LIN {X 0,Y 539.33,Z 456.687,A -85,B 0,C 180,E1 -4153.302,E2 -4153.302} C_VEL
LIN {X 0,Y 539.491,Z 386.193,A -85,B 0,C 180,E1 -4154.273,E2 -4154.273} C_VEL
LIN {X 0,Y 538.254,Z 382.203,A -85,B 0,C 180,E1 -4154.395,E2 -4154.395} C_VEL
LIN {X 0,Y 538.117,Z 381.5,A -85,B 0,C 180,E1 -4154.551,E2 -4154.551} C_VEL
LIN {X 0,Y 538.039,Z 381.463,A -85,B 0,C 180,E1 -4157.532,E2 -4157.532} C_VEL
LIN {X 0,Y 538.041,Z 381.467,A -85,B 0,C 180,E1 -4160.651,E2 -4160.651} C_VEL
LIN {X 0,Y 538.006,Z 381.464,A -85,B 0,C 180,E1 -4163.888,E2 -4163.888} C_VEL
LIN {X 0,Y 538.039,Z 381.463,A -85,B 0,C 180,E1 -4166.367,E2 -4166.367} C_VEL
LIN {X 0,Y 538.01,Z 381.462,A -85,B 0,C 180,E1 -4169.392,E2 -4169.392} C_VEL
LIN {X 0,Y 537.341,Z 381.546,A -85,B 0,C 180,E1 -4170.017,E2 -4170.017} C_VEL
LIN {X 0,Y 534.471,Z 381.909,A -85,B 0,C 180,E1 -4171.03,E2 -4171.03} C_VEL
LIN {X 0,Y 532.057,Z 382.207,A -85,B 0,C 180,E1 -4171.846,E2 -4171.846} C_VEL
LIN {X 0,Y 531.035,Z 382.338,A -85,B 0,C 180,E1 -4172.476,E2 -4172.476} C_VEL
LIN {X 0,Y 530.96,Z 382.343,A -85,B 0,C 180,E1 -4172.689,E2 -4172.689} C_VEL
LIN {X 0,Y 530.953,Z 382.342,A -85,B 0,C 180,E1 -4175.62,E2 -4175.62} C_VEL
LIN {X 0,Y 530.967,Z 382.346,A -85,B 0,C 180,E1 -4178.653,E2 -4178.653} C_VEL
LIN {X 0,Y 530.992,Z 382.337,A -85,B 0,C 180,E1 -4181.436,E2 -4181.436} C_VEL
LIN {X 0,Y 530.97,Z 382.348,A -85,B 0,C 180,E1 -4184.549,E2 -4184.549} C_VEL
LIN {X 0,Y 530.975,Z 382.34,A -85,B 0,C 180,E1 -4187.836,E2 -4187.836} C_VEL
LIN {X 0,Y 530.974,Z 382.343,A -85,B 0,C 180,E1 -4190.555,E2 -4190.555} C_VEL
LIN {X 0,Y 530.953,Z 382.344,A -85,B 0,C 180,E1 -4193.441,E2 -4193.441} C_VEL
LIN {X 0,Y 531.002,Z 382.345,A -85,B 0,C 180,E1 -4196.494,E2 -4196.494} C_VEL
LIN {X 0,Y 530.969,Z 382.342,A -85,B 0,C 180,E1 -4199.357,E2 -4199.357} C_VEL
LIN {X 0,Y 531.024,Z 382.51,A -85,B 0,C 180,E1 -4202.212,E2 -4202.212} C_VEL
LIN {X 0,Y 533.353,Z 393.17,A -85,B 0,C 180,E1 -4203.642,E2 -4203.642} C_VEL
LIN {X 0,Y 533.057,Z 413.258,A -85,B 0,C 180,E1 -4206.083,E2 -4206.083} C_VEL
LIN {X 0,Y 532.641,Z 436.75,A -85,B 0,C 180,E1 -4208.927,E2 -4208.927} C_VEL
LIN {X 0,Y 532.055,Z 463.536,A -85,B 0,C 180,E1 -4212.135,E2 -4212.135} C_VEL
LIN {X 0,Y 531.666,Z 488.086,A -85,B 0,C 180,E1 -4215.055,E2 -4215.055} C_VEL
LIN {X 0,Y 532.804,Z 497.302,A -85,B 0,C 180,E1 -4215.24,E2 -4215.24} C_VEL
LIN {X 0,Y 532.44,Z 598.014,A -85,B 0,C 180,E1 -4216.62,E2 -4216.62} C_VEL
LIN {X 0,Y 532.274,Z 610.527,A -85,B 0,C 180,E1 -4216.932,E2 -4216.932} C_VEL
LIN {X 0,Y 532.051,Z 622.317,A -85,B 0,C 180,E1 -4217.363,E2 -4217.363} C_VEL
LIN {X 0,Y 531.805,Z 635.2,A -85,B 0,C 180,E1 -4218.006,E2 -4218.006} C_VEL
LIN {X 0,Y 531.57,Z 646.587,A -85,B 0,C 180,E1 -4218.755,E2 -4218.755} C_VEL
LIN {X 0,Y 531.283,Z 655.996,A -85,B 0,C 180,E1 -4219.52,E2 -4219.52} C_VEL
LIN {X 0,Y 531.121,Z 663.859,A -85,B 0,C 180,E1 -4220.287,E2 -4220.287} C_VEL
LIN {X 0,Y 530.936,Z 670.557,A -85,B 0,C 180,E1 -4221.052,E2 -4221.052} C_VEL
LIN {X 0,Y 530.785,Z 677.606,A -85,B 0,C 180,E1 -4222.008,E2 -4222.008} C_VEL
LIN {X 0,Y 530.671,Z 683.5,A -85,B 0,C 180,E1 -4222.963,E2 -4222.963} C_VEL
LIN {X 0,Y 530.607,Z 688.403,A -85,B 0,C 180,E1 -4223.917,E2 -4223.917} C_VEL
LIN {X 0,Y 530.459,Z 693.137,A -85,B 0,C 180,E1 -4225.06,E2 -4225.06} C_VEL
LIN {X 0,Y 530.516,Z 696.771,A -85,B 0,C 180,E1 -4226.202,E2 -4226.202} C_VEL
LIN {X 0,Y 530.411,Z 700.139,A -85,B 0,C 180,E1 -4227.722,E2 -4227.722} C_VEL
LIN {X 0,Y 530.344,Z 701.716,A -85,B 0,C 180,E1 -4229.241,E2 -4229.241} C_VEL
LIN {X 0,Y 530.343,Z 701.997,A -85,B 0,C 180,E1 -4230,E2 -4230} C_VEL
LIN {X 0,Y 530.361,Z 701.19,A -85,B 0,C 180,E1 -4231.519,E2 -4231.519} C_VEL
LIN {X 0,Y 530.411,Z 700.285,A -85,B 0,C 180,E1 -4232.278,E2 -4232.278} C_VEL
LIN {X 0,Y 530.516,Z 697.021,A -85,B 0,C 180,E1 -4233.798,E2 -4233.798} C_VEL
LIN {X 0,Y 530.458,Z 693.464,A -85,B 0,C 180,E1 -4234.94,E2 -4234.94} C_VEL
LIN {X 0,Y 530.582,Z 688.812,A -85,B 0,C 180,E1 -4236.083,E2 -4236.083} C_VEL
LIN {X 0,Y 530.628,Z 683.999,A -85,B 0,C 180,E1 -4237.037,E2 -4237.037} C_VEL
LIN {X 0,Y 530.772,Z 678.202,A -85,B 0,C 180,E1 -4237.992,E2 -4237.992} C_VEL
LIN {X 0,Y 530.9,Z 671.262,A -85,B 0,C 180,E1 -4238.949,E2 -4238.949} C_VEL
LIN {X 0,Y 531.09,Z 664.693,A -85,B 0,C 180,E1 -4239.714,E2 -4239.714} C_VEL
LIN {X 0,Y 531.31,Z 655.926,A -85,B 0,C 180,E1 -4240.576,E2 -4240.576} C_VEL
LIN {X 0,Y 531.599,Z 645.228,A -85,B 0,C 180,E1 -4241.438,E2 -4241.438} C_VEL
LIN {X 0,Y 531.847,Z 633.026,A -85,B 0,C 180,E1 -4242.206,E2 -4242.206} C_VEL
LIN {X 0,Y 532.074,Z 620.98,A -85,B 0,C 180,E1 -4242.782,E2 -4242.782} C_VEL
LIN {X 0,Y 532.26,Z 608.699,A -85,B 0,C 180,E1 -4243.215,E2 -4243.215} C_VEL
LIN {X 0,Y 532.463,Z 596.37,A -85,B 0,C 180,E1 -4243.501,E2 -4243.501} C_VEL
LIN {X 0,Y 532.768,Z 496.104,A -85,B 0,C 180,E1 -4244.868,E2 -4244.868} C_VEL
LIN {X 0,Y 531.685,Z 488.274,A -85,B 0,C 180,E1 -4245.02,E2 -4245.02} C_VEL
LIN {X 0,Y 532.074,Z 463.132,A -85,B 0,C 180,E1 -4248.005,E2 -4248.005} C_VEL
LIN {X 0,Y 532.617,Z 437.549,A -85,B 0,C 180,E1 -4251.074,E2 -4251.074} C_VEL
LIN {X 0,Y 533.063,Z 414.001,A -85,B 0,C 180,E1 -4253.917,E2 -4253.917} C_VEL
LIN {X 0,Y 533.411,Z 393.872,A -85,B 0,C 180,E1 -4256.37,E2 -4256.37} C_VEL
LIN {X 0,Y 531.004,Z 382.431,A -85,B 0,C 180,E1 -4257.907,E2 -4257.907} C_VEL
LIN {X 0,Y 530.955,Z 382.348,A -85,B 0,C 180,E1 -4261.08,E2 -4261.08} C_VEL
LIN {X 0,Y 530.967,Z 382.346,A -85,B 0,C 180,E1 -4263.775,E2 -4263.775} C_VEL
LIN {X 0,Y 530.919,Z 382.344,A -85,B 0,C 180,E1 -4266.562,E2 -4266.562} C_VEL
LIN {X 0,Y 530.985,Z 382.345,A -85,B 0,C 180,E1 -4269.444,E2 -4269.444} C_VEL
LIN {X 0,Y 530.917,Z 382.348,A -85,B 0,C 180,E1 -4272.463,E2 -4272.463} C_VEL
LIN {X 0,Y 530.969,Z 382.339,A -85,B 0,C 180,E1 -4275.451,E2 -4275.451} C_VEL
LIN {X 0,Y 530.963,Z 382.341,A -85,B 0,C 180,E1 -4278.561,E2 -4278.561} C_VEL
LIN {X 0,Y 530.954,Z 382.35,A -85,B 0,C 180,E1 -4281.529,E2 -4281.529} C_VEL
LIN {X 0,Y 530.938,Z 382.345,A -85,B 0,C 180,E1 -4284.378,E2 -4284.378} C_VEL
LIN {X 0,Y 530.97,Z 382.338,A -85,B 0,C 180,E1 -4287.133,E2 -4287.133} C_VEL
LIN {X 0,Y 530.952,Z 382.348,A -85,B 0,C 180,E1 -4289.802,E2 -4289.802} C_VEL
LIN {X 0,Y 530.959,Z 382.342,A -85,B 0,C 180,E1 -4292.48,E2 -4292.48} C_VEL
LIN {X 0,Y 530.953,Z 382.342,A -85,B 0,C 180,E1 -4294.94,E2 -4294.94} C_VEL
LIN {X 0,Y 530.981,Z 382.345,A -85,B 0,C 180,E1 -4297.898,E2 -4297.898} C_VEL
LIN {X 0,Y 530.973,Z 382.338,A -85,B 0,C 180,E1 -4300.676,E2 -4300.676} C_VEL
LIN {X 0,Y 530.942,Z 382.34,A -85,B 0,C 180,E1 -4303.069,E2 -4303.069} C_VEL
LIN {X 0,Y 531.012,Z 382.34,A -85,B 0,C 180,E1 -4305.436,E2 -4305.436} C_VEL
LIN {X 0,Y 530.99,Z 382.331,A -85,B 0,C 180,E1 -4308.549,E2 -4308.549} C_VEL
LIN {X 0,Y 530.993,Z 382.344,A -85,B 0,C 180,E1 -4311.628,E2 -4311.628} C_VEL
LIN {X 0,Y 531.088,Z 382.32,A -85,B 0,C 180,E1 -4314.685,E2 -4314.685} C_VEL
LIN {X 0,Y 531.136,Z 382.325,A -85,B 0,C 180,E1 -4317.725,E2 -4317.725} C_VEL
LIN {X 0,Y 531.131,Z 382.324,A -85,B 0,C 180,E1 -4320,E2 -4320} C_VEL
LIN {X 0,Y 531.136,Z 382.315,A -85,B 0,C 180,E1 -4322.275,E2 -4322.275} C_VEL
LIN {X 0,Y 531.085,Z 382.327,A -85,B 0,C 180,E1 -4325.315,E2 -4325.315} C_VEL
LIN {X 0,Y 530.986,Z 382.335,A -85,B 0,C 180,E1 -4328.372,E2 -4328.372} C_VEL
LIN {X 0,Y 531.015,Z 382.338,A -85,B 0,C 180,E1 -4331.65,E2 -4331.65} C_VEL
LIN {X 0,Y 530.967,Z 382.339,A -85,B 0,C 180,E1 -4334.928,E2 -4334.928} C_VEL
LIN {X 0,Y 530.973,Z 382.342,A -85,B 0,C 180,E1 -4337.724,E2 -4337.724} C_VEL
LIN {X 0,Y 530.939,Z 382.343,A -85,B 0,C 180,E1 -4340.94,E2 -4340.94} C_VEL
LIN {X 0,Y 530.952,Z 382.34,A -85,B 0,C 180,E1 -4343.397,E2 -4343.397} C_VEL
LIN {X 0,Y 530.93,Z 382.353,A -85,B 0,C 180,E1 -4345.902,E2 -4345.902} C_VEL
LIN {X 0,Y 530.932,Z 382.341,A -85,B 0,C 180,E1 -4348.459,E2 -4348.459} C_VEL
LIN {X 0,Y 530.946,Z 382.343,A -85,B 0,C 180,E1 -4351.08,E2 -4351.08} C_VEL
LIN {X 0,Y 530.952,Z 382.348,A -85,B 0,C 180,E1 -4353.775,E2 -4353.775} C_VEL
LIN {X 0,Y 530.908,Z 382.349,A -85,B 0,C 180,E1 -4356.562,E2 -4356.562} C_VEL
LIN {X 0,Y 530.94,Z 382.344,A -85,B 0,C 180,E1 -4359.448,E2 -4359.448} C_VEL
LIN {X 0,Y 530.906,Z 382.344,A -85,B 0,C 180,E1 -4362.464,E2 -4362.464} C_VEL
LIN {X 0,Y 530.963,Z 382.344,A -85,B 0,C 180,E1 -4365.45,E2 -4365.45} C_VEL
LIN {X 0,Y 530.91,Z 382.337,A -85,B 0,C 180,E1 -4368.556,E2 -4368.556} C_VEL
LIN {X 0,Y 530.932,Z 382.348,A -85,B 0,C 180,E1 -4371.527,E2 -4371.527} C_VEL
LIN {X 0,Y 530.927,Z 382.35,A -85,B 0,C 180,E1 -4374.377,E2 -4374.377} C_VEL
LIN {X 0,Y 530.946,Z 382.345,A -85,B 0,C 180,E1 -4377.132,E2 -4377.132} C_VEL
LIN {X 0,Y 530.934,Z 382.353,A -85,B 0,C 180,E1 -4379.8,E2 -4379.8} C_VEL
LIN {X 0,Y 531.006,Z 382.538,A -85,B 0,C 180,E1 -4381.519,E2 -4381.519} C_VEL
LIN {X 0,Y 533.419,Z 393.223,A -85,B 0,C 180,E1 -4382.964,E2 -4382.964} C_VEL
LIN {X 0,Y 533.514,Z 400.976,A -85,B 0,C 180,E1 -4383.902,E2 -4383.902} C_VEL
LIN {X 0,Y 532.934,Z 426.254,A -85,B 0,C 180,E1 -4386.901,E2 -4386.901} C_VEL
LIN {X 0,Y 532.347,Z 450.23,A -85,B 0,C 180,E1 -4389.714,E2 -4389.714} C_VEL
LIN {X 0,Y 531.914,Z 476.387,A -85,B 0,C 180,E1 -4392.705,E2 -4392.705} C_VEL
LIN {X 0,Y 531.617,Z 496.923,A -85,B 0,C 180,E1 -4395.02,E2 -4395.02} C_VEL
LIN {X 0,Y 532.795,Z 507.185,A -85,B 0,C 180,E1 -4395.211,E2 -4395.211} C_VEL
LIN {X 0,Y 532.377,Z 607.666,A -85,B 0,C 180,E1 -4396.594,E2 -4396.594} C_VEL
LIN {X 0,Y 532.181,Z 620.892,A -85,B 0,C 180,E1 -4396.929,E2 -4396.929} C_VEL
LIN {X 0,Y 531.981,Z 633.67,A -85,B 0,C 180,E1 -4397.409,E2 -4397.409} C_VEL
LIN {X 0,Y 531.756,Z 645.607,A -85,B 0,C 180,E1 -4398.019,E2 -4398.019} C_VEL
LIN {X 0,Y 531.508,Z 656.848,A -85,B 0,C 180,E1 -4398.753,E2 -4398.753} C_VEL
LIN {X 0,Y 531.224,Z 667.468,A -85,B 0,C 180,E1 -4399.615,E2 -4399.615} C_VEL
LIN {X 0,Y 531.062,Z 676.091,A -85,B 0,C 180,E1 -4400.478,E2 -4400.478} C_VEL
LIN {X 0,Y 530.887,Z 683.959,A -85,B 0,C 180,E1 -4401.435,E2 -4401.435} C_VEL
LIN {X 0,Y 530.685,Z 691.62,A -85,B 0,C 180,E1 -4402.581,E2 -4402.581} C_VEL
LIN {X 0,Y 530.604,Z 698.678,A -85,B 0,C 180,E1 -4403.917,E2 -4403.917} C_VEL
LIN {X 0,Y 530.459,Z 703.372,A -85,B 0,C 180,E1 -4405.06,E2 -4405.06} C_VEL
LIN {X 0,Y 530.516,Z 706.957,A -85,B 0,C 180,E1 -4406.202,E2 -4406.202} C_VEL
LIN {X 0,Y 530.457,Z 708.806,A -85,B 0,C 180,E1 -4406.962,E2 -4406.962} C_VEL
LIN {X 0,Y 530.411,Z 710.193,A -85,B 0,C 180,E1 -4407.722,E2 -4407.722} C_VEL
LIN {X 0,Y 530.344,Z 711.785,A -85,B 0,C 180,E1 -4409.241,E2 -4409.241} C_VEL
LIN {X 0,Y 530.342,Z 712,A -85,B 0,C 180,E1 -4410,E2 -4410} C_VEL
LIN {X 0,Y 530.361,Z 711.183,A -85,B 0,C 180,E1 -4411.519,E2 -4411.519} C_VEL
LIN {X 0,Y 530.411,Z 710.196,A -85,B 0,C 180,E1 -4412.278,E2 -4412.278} C_VEL
LIN {X 0,Y 530.457,Z 708.81,A -85,B 0,C 180,E1 -4413.038,E2 -4413.038} C_VEL
LIN {X 0,Y 530.522,Z 705.895,A -85,B 0,C 180,E1 -4414.178,E2 -4414.178} C_VEL
LIN {X 0,Y 530.524,Z 701.948,A -85,B 0,C 180,E1 -4415.321,E2 -4415.321} C_VEL
LIN {X 0,Y 530.599,Z 696.262,A -85,B 0,C 180,E1 -4416.582,E2 -4416.582} C_VEL
LIN {X 0,Y 530.758,Z 689.235,A -85,B 0,C 180,E1 -4417.8,E2 -4417.8} C_VEL
LIN {X 0,Y 530.93,Z 680.992,A -85,B 0,C 180,E1 -4418.948,E2 -4418.948} C_VEL
LIN {X 0,Y 531.139,Z 672.486,A -85,B 0,C 180,E1 -4419.905,E2 -4419.905} C_VEL
LIN {X 0,Y 531.376,Z 661.842,A -85,B 0,C 180,E1 -4420.864,E2 -4420.864} C_VEL
LIN {X 0,Y 531.653,Z 650.613,A -85,B 0,C 180,E1 -4421.672,E2 -4421.672} C_VEL
LIN {X 0,Y 531.885,Z 639.604,A -85,B 0,C 180,E1 -4422.302,E2 -4422.302} C_VEL
LIN {X 0,Y 532.09,Z 627.599,A -85,B 0,C 180,E1 -4422.83,E2 -4422.83} C_VEL
LIN {X 0,Y 532.26,Z 613.764,A -85,B 0,C 180,E1 -4423.263,E2 -4423.263} C_VEL
LIN {X 0,Y 532.443,Z 599.688,A -85,B 0,C 180,E1 -4423.526,E2 -4423.526} C_VEL
LIN {X 0,Y 532.667,Z 505.458,A -85,B 0,C 180,E1 -4424.808,E2 -4424.808} C_VEL
LIN {X 0,Y 531.577,Z 496.346,A -85,B 0,C 180,E1 -4424.981,E2 -4424.981} C_VEL
LIN {X 0,Y 531.934,Z 469.551,A -85,B 0,C 180,E1 -4427.959,E2 -4427.959} C_VEL
LIN {X 0,Y 532.362,Z 443.563,A -85,B 0,C 180,E1 -4430.882,E2 -4430.882} C_VEL
LIN {X 0,Y 532.768,Z 416.948,A -85,B 0,C 180,E1 -4433.931,E2 -4433.931} C_VEL
LIN {X 0,Y 533.15,Z 393.927,A -85,B 0,C 180,E1 -4436.628,E2 -4436.628} C_VEL
LIN {X 0,Y 531.08,Z 383.141,A -85,B 0,C 180,E1 -4438.02,E2 -4438.02} C_VEL
LIN {X 0,Y 530.966,Z 382.478,A -85,B 0,C 180,E1 -4438.134,E2 -4438.134} C_VEL
LIN {X 0,Y 530.936,Z 382.349,A -85,B 0,C 180,E1 -4441.081,E2 -4441.081} C_VEL
LIN {X 0,Y 530.934,Z 382.353,A -85,B 0,C 180,E1 -4443.777,E2 -4443.777} C_VEL
LIN {X 0,Y 530.906,Z 382.351,A -85,B 0,C 180,E1 -4446.563,E2 -4446.563} C_VEL
LIN {X 0,Y 530.94,Z 382.349,A -85,B 0,C 180,E1 -4449.448,E2 -4449.448} C_VEL
LIN {X 0,Y 530.912,Z 382.35,A -85,B 0,C 180,E1 -4452.463,E2 -4452.463} C_VEL
LIN {X 0,Y 530.965,Z 382.347,A -85,B 0,C 180,E1 -4455.451,E2 -4455.451} C_VEL
LIN {X 0,Y 530.957,Z 382.342,A -85,B 0,C 180,E1 -4458.561,E2 -4458.561} C_VEL
LIN {X 0,Y 530.953,Z 382.351,A -85,B 0,C 180,E1 -4461.529,E2 -4461.529} C_VEL
LIN {X 0,Y 530.949,Z 382.345,A -85,B 0,C 180,E1 -4464.379,E2 -4464.379} C_VEL
LIN {X 0,Y 530.969,Z 382.345,A -85,B 0,C 180,E1 -4467.133,E2 -4467.133} C_VEL
LIN {X 0,Y 530.971,Z 382.346,A -85,B 0,C 180,E1 -4469.803,E2 -4469.803} C_VEL
LIN {X 0,Y 530.969,Z 382.341,A -85,B 0,C 180,E1 -4472.477,E2 -4472.477} C_VEL
LIN {X 0,Y 530.981,Z 382.342,A -85,B 0,C 180,E1 -4474.941,E2 -4474.941} C_VEL
LIN {X 0,Y 530.974,Z 382.342,A -85,B 0,C 180,E1 -4478.247,E2 -4478.247} C_VEL
LIN {X 0,Y 530.996,Z 382.341,A -85,B 0,C 180,E1 -4480.677,E2 -4480.677} C_VEL
LIN {X 0,Y 530.978,Z 382.348,A -85,B 0,C 180,E1 -4483.071,E2 -4483.071} C_VEL
LIN {X 0,Y 531.093,Z 382.456,A -85,B 0,C 180,E1 -4485.405,E2 -4485.405} C_VEL
LIN {X 0,Y 531.258,Z 383.232,A -85,B 0,C 180,E1 -4485.528,E2 -4485.528} C_VEL
LIN {X 0,Y 532.723,Z 388.293,A -85,B 0,C 180,E1 -4485.664,E2 -4485.664} C_VEL
LIN {X 0,Y 532.338,Z 463.302,A -85,B 0,C 180,E1 -4486.739,E2 -4486.739} C_VEL
LIN {X 0,Y 532.281,Z 476.373,A -85,B 0,C 180,E1 -4487.077,E2 -4487.077} C_VEL
LIN {X 0,Y 532.153,Z 488.956,A -85,B 0,C 180,E1 -4487.559,E2 -4487.559} C_VEL
LIN {X 0,Y 531.944,Z 500.739,A -85,B 0,C 180,E1 -4488.173,E2 -4488.173} C_VEL
LIN {X 0,Y 531.755,Z 512.234,A -85,B 0,C 180,E1 -4488.951,E2 -4488.951} C_VEL
LIN {X 0,Y 531.533,Z 522.416,A -85,B 0,C 180,E1 -4489.814,E2 -4489.814} C_VEL
LIN {X 0,Y 531.339,Z 530.703,A -85,B 0,C 180,E1 -4490.675,E2 -4490.675} C_VEL
LIN {X 0,Y 531.143,Z 539.63,A -85,B 0,C 180,E1 -4491.822,E2 -4491.822} C_VEL
LIN {X 0,Y 531.01,Z 545.698,A -85,B 0,C 180,E1 -4492.777,E2 -4492.777} C_VEL
LIN {X 0,Y 530.92,Z 551.605,A -85,B 0,C 180,E1 -4493.921,E2 -4493.921} C_VEL
LIN {X 0,Y 530.758,Z 556.277,A -85,B 0,C 180,E1 -4495.062,E2 -4495.062} C_VEL
LIN {X 0,Y 530.707,Z 559.862,A -85,B 0,C 180,E1 -4496.203,E2 -4496.203} C_VEL
LIN {X 0,Y 530.688,Z 561.676,A -85,B 0,C 180,E1 -4496.963,E2 -4496.963} C_VEL
LIN {X 0,Y 530.612,Z 563.086,A -85,B 0,C 180,E1 -4497.723,E2 -4497.723} C_VEL
LIN {X 0,Y 530.593,Z 564.638,A -85,B 0,C 180,E1 -4499.241,E2 -4499.241} C_VEL
LIN {X 0,Y 530.583,Z 564.855,A -85,B 0,C 180,E1 -4500,E2 -4500} C_VEL
LIN {X 0,Y 530.575,Z 564.046,A -85,B 0,C 180,E1 -4501.518,E2 -4501.518} C_VEL
LIN {X 0,Y 530.607,Z 563.084,A -85,B 0,C 180,E1 -4502.277,E2 -4502.277} C_VEL
LIN {X 0,Y 530.643,Z 561.706,A -85,B 0,C 180,E1 -4503.037,E2 -4503.037} C_VEL
LIN {X 0,Y 530.709,Z 557.643,A -85,B 0,C 180,E1 -4504.557,E2 -4504.557} C_VEL
LIN {X 0,Y 530.811,Z 553.379,A -85,B 0,C 180,E1 -4505.699,E2 -4505.699} C_VEL
LIN {X 0,Y 530.884,Z 547.935,A -85,B 0,C 180,E1 -4506.843,E2 -4506.843} C_VEL
LIN {X 0,Y 531.03,Z 541.097,A -85,B 0,C 180,E1 -4507.988,E2 -4507.988} C_VEL
LIN {X 0,Y 531.24,Z 534.11,A -85,B 0,C 180,E1 -4508.943,E2 -4508.943} C_VEL
LIN {X 0,Y 531.382,Z 525.669,A -85,B 0,C 180,E1 -4509.901,E2 -4509.901} C_VEL
LIN {X 0,Y 531.633,Z 515.231,A -85,B 0,C 180,E1 -4510.858,E2 -4510.858} C_VEL
LIN {X 0,Y 531.924,Z 503.763,A -85,B 0,C 180,E1 -4511.695,E2 -4511.695} C_VEL
LIN {X 0,Y 532.036,Z 493.307,A -85,B 0,C 180,E1 -4512.299,E2 -4512.299} C_VEL
LIN {X 0,Y 532.194,Z 481.358,A -85,B 0,C 180,E1 -4512.828,E2 -4512.828} C_VEL
LIN {X 0,Y 532.31,Z 468.412,A -85,B 0,C 180,E1 -4513.238,E2 -4513.238} C_VEL
LIN {X 0,Y 532.418,Z 454.629,A -85,B 0,C 180,E1 -4513.502,E2 -4513.502} C_VEL
LIN {X 0,Y 532.598,Z 387.511,A -85,B 0,C 180,E1 -4514.443,E2 -4514.443} C_VEL
LIN {X 0,Y 531.213,Z 383.1,A -85,B 0,C 180,E1 -4514.575,E2 -4514.575} C_VEL
LIN {X 0,Y 531.049,Z 382.389,A -85,B 0,C 180,E1 -4514.729,E2 -4514.729} C_VEL
LIN {X 0,Y 530.985,Z 382.341,A -85,B 0,C 180,E1 -4517.724,E2 -4517.724} C_VEL
LIN {X 0,Y 531.028,Z 382.336,A -85,B 0,C 180,E1 -4520.127,E2 -4520.127} C_VEL
LIN {X 0,Y 530.949,Z 382.35,A -85,B 0,C 180,E1 -4522.573,E2 -4522.573} C_VEL
LIN {X 0,Y 531.002,Z 382.341,A -85,B 0,C 180,E1 -4525.058,E2 -4525.058} C_VEL
LIN {X 0,Y 530.973,Z 382.338,A -85,B 0,C 180,E1 -4527.598,E2 -4527.598} C_VEL
LIN {X 0,Y 530.972,Z 382.34,A -85,B 0,C 180,E1 -4530.197,E2 -4530.197} C_VEL
LIN {X 0,Y 530.96,Z 382.343,A -85,B 0,C 180,E1 -4532.689,E2 -4532.689} C_VEL
LIN {X 0,Y 530.309,Z 382.426,A -85,B 0,C 180,E1 -4533.322,E2 -4533.322} C_VEL
LIN {X 0,Y 527.435,Z 382.783,A -85,B 0,C 180,E1 -4534.349,E2 -4534.349} C_VEL
LIN {X 0,Y 525.002,Z 383.086,A -85,B 0,C 180,E1 -4535.176,E2 -4535.176} C_VEL
LIN {X 0,Y 523.969,Z 383.213,A -85,B 0,C 180,E1 -4535.816,E2 -4535.816} C_VEL
LIN {X 0,Y 523.893,Z 383.223,A -85,B 0,C 180,E1 -4536.032,E2 -4536.032} C_VEL
LIN {X 0,Y 523.922,Z 383.222,A -85,B 0,C 180,E1 -4539.085,E2 -4539.085} C_VEL
LIN {X 0,Y 523.943,Z 383.216,A -85,B 0,C 180,E1 -4542.12,E2 -4542.12} C_VEL
LIN {X 0,Y 523.943,Z 383.216,A -85,B 0,C 180,E1 -4545.311,E2 -4545.311} C_VEL
LIN {X 0,Y 523.956,Z 383.222,A -85,B 0,C 180,E1 -4548.69,E2 -4548.69} C_VEL
LIN {X 0,Y 523.915,Z 383.215,A -85,B 0,C 180,E1 -4551.898,E2 -4551.898} C_VEL
LIN {X 0,Y 523.925,Z 383.219,A -85,B 0,C 180,E1 -4554.912,E2 -4554.912} C_VEL
LIN {X 0,Y 523.938,Z 383.215,A -85,B 0,C 180,E1 -4557.68,E2 -4557.68} C_VEL
LIN {X 0,Y 523.955,Z 383.223,A -85,B 0,C 180,E1 -4560.677,E2 -4560.677} C_VEL
LIN {X 0,Y 523.987,Z 383.416,A -85,B 0,C 180,E1 -4562.002,E2 -4562.002} C_VEL
LIN {X 0,Y 526.586,Z 395.433,A -85,B 0,C 180,E1 -4563.615,E2 -4563.615} C_VEL
LIN {X 0,Y 526.099,Z 419.563,A -85,B 0,C 180,E1 -4566.583,E2 -4566.583} C_VEL
LIN {X 0,Y 525.542,Z 443.703,A -85,B 0,C 180,E1 -4569.527,E2 -4569.527} C_VEL
LIN {X 0,Y 525.009,Z 468.06,A -85,B 0,C 180,E1 -4572.471,E2 -4572.471} C_VEL
LIN {X 0,Y 524.739,Z 488.377,A -85,B 0,C 180,E1 -4574.873,E2 -4574.873} C_VEL
LIN {X 0,Y 525.966,Z 498.434,A -85,B 0,C 180,E1 -4575.059,E2 -4575.059} C_VEL
LIN {X 0,Y 525.54,Z 597.969,A -85,B 0,C 180,E1 -4576.441,E2 -4576.441} C_VEL
LIN {X 0,Y 525.372,Z 610.614,A -85,B 0,C 180,E1 -4576.757,E2 -4576.757} C_VEL
LIN {X 0,Y 525.091,Z 623.487,A -85,B 0,C 180,E1 -4577.242,E2 -4577.242} C_VEL
LIN {X 0,Y 524.827,Z 636.17,A -85,B 0,C 180,E1 -4577.9,E2 -4577.9} C_VEL
LIN {X 0,Y 524.605,Z 646.702,A -85,B 0,C 180,E1 -4578.603,E2 -4578.603} C_VEL
LIN {X 0,Y 524.274,Z 657.16,A -85,B 0,C 180,E1 -4579.476,E2 -4579.476} C_VEL
LIN {X 0,Y 524.004,Z 667.467,A -85,B 0,C 180,E1 -4580.544,E2 -4580.544} C_VEL
LIN {X 0,Y 523.767,Z 676.422,A -85,B 0,C 180,E1 -4581.706,E2 -4581.706} C_VEL
LIN {X 0,Y 523.61,Z 683.596,A -85,B 0,C 180,E1 -4582.868,E2 -4582.868} C_VEL
LIN {X 0,Y 523.518,Z 688.478,A -85,B 0,C 180,E1 -4583.835,E2 -4583.835} C_VEL
LIN {X 0,Y 523.383,Z 693.192,A -85,B 0,C 180,E1 -4584.993,E2 -4584.993} C_VEL
LIN {X 0,Y 523.443,Z 696.815,A -85,B 0,C 180,E1 -4586.151,E2 -4586.151} C_VEL
LIN {X 0,Y 523.368,Z 698.695,A -85,B 0,C 180,E1 -4586.921,E2 -4586.921} C_VEL
LIN {X 0,Y 523.335,Z 700.161,A -85,B 0,C 180,E1 -4587.691,E2 -4587.691} C_VEL
LIN {X 0,Y 523.25,Z 701.746,A -85,B 0,C 180,E1 -4589.231,E2 -4589.231} C_VEL
LIN {X 0,Y 523.247,Z 702.013,A -85,B 0,C 180,E1 -4590,E2 -4590} C_VEL
LIN {X 0,Y 523.275,Z 701.22,A -85,B 0,C 180,E1 -4591.539,E2 -4591.539} C_VEL
LIN {X 0,Y 523.335,Z 700.298,A -85,B 0,C 180,E1 -4592.309,E2 -4592.309} C_VEL
LIN {X 0,Y 523.444,Z 697.06,A -85,B 0,C 180,E1 -4593.849,E2 -4593.849} C_VEL
LIN {X 0,Y 523.383,Z 693.514,A -85,B 0,C 180,E1 -4595.007,E2 -4595.007} C_VEL
LIN {X 0,Y 523.495,Z 688.88,A -85,B 0,C 180,E1 -4596.166,E2 -4596.166} C_VEL
LIN {X 0,Y 523.596,Z 683.021,A -85,B 0,C 180,E1 -4597.326,E2 -4597.326} C_VEL
LIN {X 0,Y 523.78,Z 675.711,A -85,B 0,C 180,E1 -4598.488,E2 -4598.488} C_VEL
LIN {X 0,Y 524.029,Z 666.542,A -85,B 0,C 180,E1 -4599.651,E2 -4599.651} C_VEL
LIN {X 0,Y 524.269,Z 657.083,A -85,B 0,C 180,E1 -4600.622,E2 -4600.622} C_VEL
LIN {X 0,Y 524.584,Z 646.593,A -85,B 0,C 180,E1 -4601.495,E2 -4601.495} C_VEL
LIN {X 0,Y 524.858,Z 635.031,A -85,B 0,C 180,E1 -4602.256,E2 -4602.256} C_VEL
LIN {X 0,Y 525.136,Z 623.309,A -85,B 0,C 180,E1 -4602.856,E2 -4602.856} C_VEL
LIN {X 0,Y 525.322,Z 610.329,A -85,B 0,C 180,E1 -4603.343,E2 -4603.343} C_VEL
LIN {X 0,Y 525.576,Z 596.262,A -85,B 0,C 180,E1 -4603.681,E2 -4603.681} C_VEL
LIN {X 0,Y 525.839,Z 496.381,A -85,B 0,C 180,E1 -4605.063,E2 -4605.063} C_VEL
LIN {X 0,Y 524.739,Z 488.223,A -85,B 0,C 180,E1 -4605.225,E2 -4605.225} C_VEL
LIN {X 0,Y 525.111,Z 463.755,A -85,B 0,C 180,E1 -4608.148,E2 -4608.148} C_VEL
LIN {X 0,Y 525.661,Z 438.795,A -85,B 0,C 180,E1 -4611.161,E2 -4611.161} C_VEL
LIN {X 0,Y 526.17,Z 415.264,A -85,B 0,C 180,E1 -4614.041,E2 -4614.041} C_VEL
LIN {X 0,Y 526.588,Z 395.96,A -85,B 0,C 180,E1 -4616.417,E2 -4616.417} C_VEL
LIN {X 0,Y 524.406,Z 385.405,A -85,B 0,C 180,E1 -4617.807,E2 -4617.807} C_VEL
LIN {X 0,Y 523.943,Z 383.28,A -85,B 0,C 180,E1 -4618.137,E2 -4618.137} C_VEL
LIN {X 0,Y 523.939,Z 383.22,A -85,B 0,C 180,E1 -4620.853,E2 -4620.853} C_VEL
LIN {X 0,Y 523.943,Z 383.221,A -85,B 0,C 180,E1 -4623.731,E2 -4623.731} C_VEL
LIN {X 0,Y 523.871,Z 383.223,A -85,B 0,C 180,E1 -4626.396,E2 -4626.396} C_VEL
LIN {X 0,Y 523.92,Z 383.222,A -85,B 0,C 180,E1 -4629.085,E2 -4629.085} C_VEL
LIN {X 0,Y 523.898,Z 383.225,A -85,B 0,C 180,E1 -4632.125,E2 -4632.125} C_VEL
LIN {X 0,Y 523.939,Z 383.213,A -85,B 0,C 180,E1 -4635.311,E2 -4635.311} C_VEL
LIN {X 0,Y 523.924,Z 383.218,A -85,B 0,C 180,E1 -4638.694,E2 -4638.694} C_VEL
LIN {X 0,Y 523.906,Z 383.223,A -85,B 0,C 180,E1 -4641.897,E2 -4641.897} C_VEL
LIN {X 0,Y 523.918,Z 383.219,A -85,B 0,C 180,E1 -4644.913,E2 -4644.913} C_VEL
LIN {X 0,Y 523.939,Z 383.222,A -85,B 0,C 180,E1 -4647.68,E2 -4647.68} C_VEL
LIN {X 0,Y 523.939,Z 383.213,A -85,B 0,C 180,E1 -4650.681,E2 -4650.681} C_VEL
LIN {X 0,Y 523.901,Z 383.23,A -85,B 0,C 180,E1 -4653.724,E2 -4653.724} C_VEL
LIN {X 0,Y 523.913,Z 383.217,A -85,B 0,C 180,E1 -4656.269,E2 -4656.269} C_VEL
LIN {X 0,Y 523.945,Z 383.215,A -85,B 0,C 180,E1 -4658.766,E2 -4658.766} C_VEL
LIN {X 0,Y 523.933,Z 383.218,A -85,B 0,C 180,E1 -4661.22,E2 -4661.22} C_VEL
LIN {X 0,Y 523.886,Z 383.226,A -85,B 0,C 180,E1 -4663.637,E2 -4663.637} C_VEL
LIN {X 0,Y 523.928,Z 383.221,A -85,B 0,C 180,E1 -4666.028,E2 -4666.028} C_VEL
LIN {X 0,Y 523.964,Z 383.207,A -85,B 0,C 180,E1 -4668.393,E2 -4668.393} C_VEL
LIN {X 0,Y 523.956,Z 383.218,A -85,B 0,C 180,E1 -4671.515,E2 -4671.515} C_VEL
LIN {X 0,Y 524.035,Z 383.199,A -85,B 0,C 180,E1 -4674.613,E2 -4674.613} C_VEL
LIN {X 0,Y 524.107,Z 383.2,A -85,B 0,C 180,E1 -4677.694,E2 -4677.694} C_VEL
LIN {X 0,Y 524.1,Z 383.199,A -85,B 0,C 180,E1 -4680,E2 -4680} C_VEL
LIN {X 0,Y 524.106,Z 383.19,A -85,B 0,C 180,E1 -4682.306,E2 -4682.306} C_VEL
LIN {X 0,Y 524.004,Z 383.211,A -85,B 0,C 180,E1 -4686.16,E2 -4686.16} C_VEL
LIN {X 0,Y 523.947,Z 383.212,A -85,B 0,C 180,E1 -4689.263,E2 -4689.263} C_VEL
LIN {X 0,Y 523.95,Z 383.216,A -85,B 0,C 180,E1 -4692.393,E2 -4692.393} C_VEL
LIN {X 0,Y 523.885,Z 383.226,A -85,B 0,C 180,E1 -4695.563,E2 -4695.563} C_VEL
LIN {X 0,Y 523.908,Z 383.226,A -85,B 0,C 180,E1 -4697.971,E2 -4697.971} C_VEL
LIN {X 0,Y 523.909,Z 383.221,A -85,B 0,C 180,E1 -4700.413,E2 -4700.413} C_VEL
LIN {X 0,Y 523.91,Z 383.214,A -85,B 0,C 180,E1 -4702.894,E2 -4702.894} C_VEL
LIN {X 0,Y 523.881,Z 383.225,A -85,B 0,C 180,E1 -4705.422,E2 -4705.422} C_VEL
LIN {X 0,Y 523.898,Z 383.223,A -85,B 0,C 180,E1 -4708.003,E2 -4708.003} C_VEL
LIN {X 0,Y 523.911,Z 383.219,A -85,B 0,C 180,E1 -4710.848,E2 -4710.848} C_VEL
LIN {X 0,Y 523.928,Z 383.223,A -85,B 0,C 180,E1 -4713.729,E2 -4713.729} C_VEL
LIN {X 0,Y 523.862,Z 383.228,A -85,B 0,C 180,E1 -4716.394,E2 -4716.394} C_VEL
LIN {X 0,Y 523.895,Z 383.219,A -85,B 0,C 180,E1 -4719.087,E2 -4719.087} C_VEL
LIN {X 0,Y 523.888,Z 383.217,A -85,B 0,C 180,E1 -4722.125,E2 -4722.125} C_VEL
LIN {X 0,Y 523.934,Z 383.218,A -85,B 0,C 180,E1 -4725.311,E2 -4725.311} C_VEL
LIN {X 0,Y 523.878,Z 383.211,A -85,B 0,C 180,E1 -4728.7,E2 -4728.7} C_VEL
LIN {X 0,Y 523.89,Z 383.231,A -85,B 0,C 180,E1 -4731.896,E2 -4731.896} C_VEL
LIN {X 0,Y 523.89,Z 383.224,A -85,B 0,C 180,E1 -4734.917,E2 -4734.917} C_VEL
LIN {X 0,Y 523.9,Z 383.229,A -85,B 0,C 180,E1 -4737.686,E2 -4737.686} C_VEL
LIN {X 0,Y 523.869,Z 383.233,A -85,B 0,C 180,E1 -4740.239,E2 -4740.239} C_VEL
LIN {X 0,Y 523.962,Z 383.42,A -85,B 0,C 180,E1 -4741.292,E2 -4741.292} C_VEL
LIN {X 0,Y 526.708,Z 396.065,A -85,B 0,C 180,E1 -4743.02,E2 -4743.02} C_VEL
LIN {X 0,Y 526.319,Z 414.38,A -85,B 0,C 180,E1 -4745.233,E2 -4745.233} C_VEL
LIN {X 0,Y 525.737,Z 437.567,A -85,B 0,C 180,E1 -4748.019,E2 -4748.019} C_VEL
LIN {X 0,Y 525.169,Z 461.75,A -85,B 0,C 180,E1 -4750.86,E2 -4750.86} C_VEL
LIN {X 0,Y 524.72,Z 486.034,A -85,B 0,C 180,E1 -4753.664,E2 -4753.664} C_VEL
LIN {X 0,Y 524.613,Z 496.029,A -85,B 0,C 180,E1 -4754.811,E2 -4754.811} C_VEL
LIN {X 0,Y 525.912,Z 508.101,A -85,B 0,C 180,E1 -4755.039,E2 -4755.039} C_VEL
LIN {X 0,Y 525.436,Z 607.186,A -85,B 0,C 180,E1 -4756.438,E2 -4756.438} C_VEL
LIN {X 0,Y 525.218,Z 620.255,A -85,B 0,C 180,E1 -4756.777,E2 -4756.777} C_VEL
LIN {X 0,Y 524.997,Z 632.385,A -85,B 0,C 180,E1 -4757.239,E2 -4757.239} C_VEL
LIN {X 0,Y 524.737,Z 644.868,A -85,B 0,C 180,E1 -4757.883,E2 -4757.883} C_VEL
LIN {X 0,Y 524.44,Z 657.035,A -85,B 0,C 180,E1 -4758.697,E2 -4758.697} C_VEL
LIN {X 0,Y 524.141,Z 667.463,A -85,B 0,C 180,E1 -4759.571,E2 -4759.571} C_VEL
LIN {X 0,Y 523.941,Z 676.848,A -85,B 0,C 180,E1 -4760.542,E2 -4760.542} C_VEL
LIN {X 0,Y 523.76,Z 685.995,A -85,B 0,C 180,E1 -4761.706,E2 -4761.706} C_VEL
LIN {X 0,Y 523.584,Z 693.347,A -85,B 0,C 180,E1 -4762.868,E2 -4762.868} C_VEL
LIN {X 0,Y 523.496,Z 698.324,A -85,B 0,C 180,E1 -4763.834,E2 -4763.834} C_VEL
LIN {X 0,Y 523.383,Z 703.151,A -85,B 0,C 180,E1 -4764.993,E2 -4764.993} C_VEL
LIN {X 0,Y 523.443,Z 706.845,A -85,B 0,C 180,E1 -4766.151,E2 -4766.151} C_VEL
LIN {X 0,Y 523.367,Z 708.726,A -85,B 0,C 180,E1 -4766.921,E2 -4766.921} C_VEL
LIN {X 0,Y 523.335,Z 710.135,A -85,B 0,C 180,E1 -4767.691,E2 -4767.691} C_VEL
LIN {X 0,Y 523.25,Z 711.747,A -85,B 0,C 180,E1 -4769.23,E2 -4769.23} C_VEL
LIN {X 0,Y 523.246,Z 711.964,A -85,B 0,C 180,E1 -4770,E2 -4770} C_VEL
LIN {X 0,Y 523.274,Z 711.138,A -85,B 0,C 180,E1 -4771.539,E2 -4771.539} C_VEL
LIN {X 0,Y 523.335,Z 710.139,A -85,B 0,C 180,E1 -4772.309,E2 -4772.309} C_VEL
LIN {X 0,Y 523.367,Z 708.73,A -85,B 0,C 180,E1 -4773.079,E2 -4773.079} C_VEL
LIN {X 0,Y 523.425,Z 705.755,A -85,B 0,C 180,E1 -4774.235,E2 -4774.235} C_VEL
LIN {X 0,Y 523.464,Z 701.692,A -85,B 0,C 180,E1 -4775.393,E2 -4775.393} C_VEL
LIN {X 0,Y 523.523,Z 696.289,A -85,B 0,C 180,E1 -4776.581,E2 -4776.581} C_VEL
LIN {X 0,Y 523.665,Z 689.82,A -85,B 0,C 180,E1 -4777.713,E2 -4777.713} C_VEL
LIN {X 0,Y 523.845,Z 681.569,A -85,B 0,C 180,E1 -4778.875,E2 -4778.875} C_VEL
LIN {X 0,Y 524.054,Z 673.155,A -85,B 0,C 180,E1 -4779.845,E2 -4779.845} C_VEL
LIN {X 0,Y 524.274,Z 662.877,A -85,B 0,C 180,E1 -4780.817,E2 -4780.817} C_VEL
LIN {X 0,Y 524.576,Z 651.172,A -85,B 0,C 180,E1 -4781.697,E2 -4781.697} C_VEL
LIN {X 0,Y 524.83,Z 639.879,A -85,B 0,C 180,E1 -4782.372,E2 -4782.372} C_VEL
LIN {X 0,Y 525.037,Z 628.383,A -85,B 0,C 180,E1 -4782.907,E2 -4782.907} C_VEL
LIN {X 0,Y 525.253,Z 615.482,A -85,B 0,C 180,E1 -4783.345,E2 -4783.345} C_VEL
LIN {X 0,Y 525.49,Z 601.971,A -85,B 0,C 180,E1 -4783.634,E2 -4783.634} C_VEL
LIN {X 0,Y 525.739,Z 505.857,A -85,B 0,C 180,E1 -4784.982,E2 -4784.982} C_VEL
LIN {X 0,Y 524.536,Z 495.222,A -85,B 0,C 180,E1 -4785.179,E2 -4785.179} C_VEL
LIN {X 0,Y 524.927,Z 468.259,A -85,B 0,C 180,E1 -4788.216,E2 -4788.216} C_VEL
LIN {X 0,Y 525.365,Z 440.605,A -85,B 0,C 180,E1 -4791.379,E2 -4791.379} C_VEL
LIN {X 0,Y 525.89,Z 414.079,A -85,B 0,C 180,E1 -4794.474,E2 -4794.474} C_VEL
LIN {X 0,Y 526.159,Z 394.224,A -85,B 0,C 180,E1 -4796.856,E2 -4796.856} C_VEL
LIN {X 0,Y 523.904,Z 383.36,A -85,B 0,C 180,E1 -4798.33,E2 -4798.33} C_VEL
LIN {X 0,Y 523.905,Z 383.227,A -85,B 0,C 180,E1 -4801.545,E2 -4801.545} C_VEL
LIN {X 0,Y 523.904,Z 383.227,A -85,B 0,C 180,E1 -4804.293,E2 -4804.293} C_VEL
LIN {X 0,Y 523.873,Z 383.232,A -85,B 0,C 180,E1 -4807.673,E2 -4807.673} C_VEL
LIN {X 0,Y 523.883,Z 383.229,A -85,B 0,C 180,E1 -4810.122,E2 -4810.122} C_VEL
LIN {X 0,Y 523.88,Z 383.227,A -85,B 0,C 180,E1 -4813.171,E2 -4813.171} C_VEL
LIN {X 0,Y 523.92,Z 383.227,A -85,B 0,C 180,E1 -4815.77,E2 -4815.77} C_VEL
LIN {X 0,Y 523.895,Z 383.223,A -85,B 0,C 180,E1 -4818.903,E2 -4818.903} C_VEL
LIN {X 0,Y 523.905,Z 383.227,A -85,B 0,C 180,E1 -4821.897,E2 -4821.897} C_VEL
LIN {X 0,Y 523.922,Z 383.221,A -85,B 0,C 180,E1 -4824.912,E2 -4824.912} C_VEL
LIN {X 0,Y 523.937,Z 383.224,A -85,B 0,C 180,E1 -4827.68,E2 -4827.68} C_VEL
LIN {X 0,Y 523.955,Z 383.216,A -85,B 0,C 180,E1 -4830.677,E2 -4830.677} C_VEL
LIN {X 0,Y 523.93,Z 383.223,A -85,B 0,C 180,E1 -4833.726,E2 -4833.726} C_VEL
LIN {X 0,Y 523.914,Z 383.221,A -85,B 0,C 180,E1 -4836.27,E2 -4836.27} C_VEL
LIN {X 0,Y 523.949,Z 383.218,A -85,B 0,C 180,E1 -4838.767,E2 -4838.767} C_VEL
LIN {X 0,Y 523.951,Z 383.223,A -85,B 0,C 180,E1 -4841.221,E2 -4841.221} C_VEL
LIN {X 0,Y 523.935,Z 383.225,A -85,B 0,C 180,E1 -4843.639,E2 -4843.639} C_VEL
LIN {X 0,Y 524.028,Z 383.421,A -85,B 0,C 180,E1 -4845.237,E2 -4845.237} C_VEL
LIN {X 0,Y 524.272,Z 384.411,A -85,B 0,C 180,E1 -4845.356,E2 -4845.356} C_VEL
LIN {X 0,Y 525.84,Z 389.274,A -85,B 0,C 180,E1 -4845.487,E2 -4845.487} C_VEL
LIN {X 0,Y 525.445,Z 465.445,A -85,B 0,C 180,E1 -4846.611,E2 -4846.611} C_VEL
LIN {X 0,Y 525.354,Z 478.921,A -85,B 0,C 180,E1 -4846.978,E2 -4846.978} C_VEL
LIN {X 0,Y 525.251,Z 490.559,A -85,B 0,C 180,E1 -4847.442,E2 -4847.442} C_VEL
LIN {X 0,Y 525.033,Z 501.697,A -85,B 0,C 180,E1 -4848.032,E2 -4848.032} C_VEL
LIN {X 0,Y 524.85,Z 513.006,A -85,B 0,C 180,E1 -4848.804,E2 -4848.804} C_VEL
LIN {X 0,Y 524.606,Z 523.255,A -85,B 0,C 180,E1 -4849.678,E2 -4849.678} C_VEL
LIN {X 0,Y 524.398,Z 531.595,A -85,B 0,C 180,E1 -4850.551,E2 -4850.551} C_VEL
LIN {X 0,Y 524.184,Z 540.573,A -85,B 0,C 180,E1 -4851.713,E2 -4851.713} C_VEL
LIN {X 0,Y 524.04,Z 546.672,A -85,B 0,C 180,E1 -4852.681,E2 -4852.681} C_VEL
LIN {X 0,Y 523.943,Z 552.604,A -85,B 0,C 180,E1 -4853.84,E2 -4853.84} C_VEL
LIN {X 0,Y 523.769,Z 557.293,A -85,B 0,C 180,E1 -4854.996,E2 -4854.996} C_VEL
LIN {X 0,Y 523.694,Z 560.869,A -85,B 0,C 180,E1 -4856.153,E2 -4856.153} C_VEL
LIN {X 0,Y 523.697,Z 562.695,A -85,B 0,C 180,E1 -4856.923,E2 -4856.923} C_VEL
LIN {X 0,Y 523.605,Z 564.098,A -85,B 0,C 180,E1 -4857.692,E2 -4857.692} C_VEL
LIN {X 0,Y 523.582,Z 565.647,A -85,B 0,C 180,E1 -4859.231,E2 -4859.231} C_VEL
LIN {X 0,Y 523.57,Z 565.857,A -85,B 0,C 180,E1 -4860,E2 -4860} C_VEL
LIN {X 0,Y 523.581,Z 565.65,A -85,B 0,C 180,E1 -4860.769,E2 -4860.769} C_VEL
LIN {X 0,Y 523.599,Z 564.049,A -85,B 0,C 180,E1 -4862.308,E2 -4862.308} C_VEL
LIN {X 0,Y 523.618,Z 562.667,A -85,B 0,C 180,E1 -4863.078,E2 -4863.078} C_VEL
LIN {X 0,Y 523.724,Z 559.751,A -85,B 0,C 180,E1 -4864.233,E2 -4864.233} C_VEL
LIN {X 0,Y 523.73,Z 555.841,A -85,B 0,C 180,E1 -4865.39,E2 -4865.39} C_VEL
LIN {X 0,Y 523.884,Z 550.184,A -85,B 0,C 180,E1 -4866.666,E2 -4866.666} C_VEL
LIN {X 0,Y 524.024,Z 543.167,A -85,B 0,C 180,E1 -4867.901,E2 -4867.901} C_VEL
LIN {X 0,Y 524.291,Z 534.907,A -85,B 0,C 180,E1 -4869.062,E2 -4869.062} C_VEL
LIN {X 0,Y 524.437,Z 526.413,A -85,B 0,C 180,E1 -4870.033,E2 -4870.033} C_VEL
LIN {X 0,Y 524.708,Z 515.88,A -85,B 0,C 180,E1 -4871.003,E2 -4871.003} C_VEL
LIN {X 0,Y 525.006,Z 504.556,A -85,B 0,C 180,E1 -4871.837,E2 -4871.837} C_VEL
LIN {X 0,Y 525.133,Z 493.793,A -85,B 0,C 180,E1 -4872.463,E2 -4872.463} C_VEL
LIN {X 0,Y 525.281,Z 481.703,A -85,B 0,C 180,E1 -4873,E2 -4873} C_VEL
LIN {X 0,Y 525.412,Z 468.528,A -85,B 0,C 180,E1 -4873.415,E2 -4873.415} C_VEL
LIN {X 0,Y 525.519,Z 455.77,A -85,B 0,C 180,E1 -4873.658,E2 -4873.658} C_VEL
LIN {X 0,Y 525.682,Z 388.8,A -85,B 0,C 180,E1 -4874.618,E2 -4874.618} C_VEL
LIN {X 0,Y 524.145,Z 384.03,A -85,B 0,C 180,E1 -4874.76,E2 -4874.76} C_VEL
LIN {X 0,Y 524.017,Z 383.262,A -85,B 0,C 180,E1 -4874.927,E2 -4874.927} C_VEL
LIN {X 0,Y 523.951,Z 383.218,A -85,B 0,C 180,E1 -4877.97,E2 -4877.97} C_VEL
LIN {X 0,Y 523.975,Z 383.217,A -85,B 0,C 180,E1 -4880.41,E2 -4880.41} C_VEL
LIN {X 0,Y 523.914,Z 383.227,A -85,B 0,C 180,E1 -4882.894,E2 -4882.894} C_VEL
LIN {X 0,Y 523.938,Z 383.217,A -85,B 0,C 180,E1 -4885.42,E2 -4885.42} C_VEL
LIN {X 0,Y 523.921,Z 383.216,A -85,B 0,C 180,E1 -4888.002,E2 -4888.002} C_VEL
LIN {X 0,Y 523.948,Z 383.223,A -85,B 0,C 180,E1 -4890.855,E2 -4890.855} C_VEL
LIN {X 0,Y 523.933,Z 383.212,A -85,B 0,C 180,E1 -4893.73,E2 -4893.73} C_VEL
LIN {X 0,Y 523.893,Z 383.223,A -85,B 0,C 180,E1 -4896.032,E2 -4896.032} C_VEL
LIN {X 0,Y 523.248,Z 383.31,A -85,B 0,C 180,E1 -4896.674,E2 -4896.674} C_VEL
LIN {X 0,Y 520.41,Z 383.663,A -85,B 0,C 180,E1 -4897.715,E2 -4897.715} C_VEL
LIN {X 0,Y 517.999,Z 383.961,A -85,B 0,C 180,E1 -4898.554,E2 -4898.554} C_VEL
LIN {X 0,Y 516.964,Z 384.088,A -85,B 0,C 180,E1 -4899.202,E2 -4899.202} C_VEL
LIN {X 0,Y 516.881,Z 384.096,A -85,B 0,C 180,E1 -4899.422,E2 -4899.422} C_VEL
LIN {X 0,Y 516.909,Z 384.091,A -85,B 0,C 180,E1 -4901.776,E2 -4901.776} C_VEL
LIN {X 0,Y 516.898,Z 384.096,A -85,B 0,C 180,E1 -4905.007,E2 -4905.007} C_VEL
LIN {X 0,Y 516.912,Z 384.096,A -85,B 0,C 180,E1 -4908.399,E2 -4908.399} C_VEL
LIN {X 0,Y 516.879,Z 384.09,A -85,B 0,C 180,E1 -4911.284,E2 -4911.284} C_VEL
LIN {X 0,Y 516.87,Z 384.103,A -85,B 0,C 180,E1 -4914.219,E2 -4914.219} C_VEL
LIN {X 0,Y 516.897,Z 384.094,A -85,B 0,C 180,E1 -4917.053,E2 -4917.053} C_VEL
LIN {X 0,Y 516.889,Z 384.096,A -85,B 0,C 180,E1 -4919.796,E2 -4919.796} C_VEL
LIN {X 0,Y 516.964,Z 384.279,A -85,B 0,C 180,E1 -4921.779,E2 -4921.779} C_VEL
LIN {X 0,Y 519.733,Z 396.951,A -85,B 0,C 180,E1 -4923.497,E2 -4923.497} C_VEL
LIN {X 0,Y 519.266,Z 419.157,A -85,B 0,C 180,E1 -4926.256,E2 -4926.256} C_VEL
LIN {X 0,Y 518.621,Z 444.355,A -85,B 0,C 180,E1 -4929.37,E2 -4929.37} C_VEL
LIN {X 0,Y 518.049,Z 469.535,A -85,B 0,C 180,E1 -4932.431,E2 -4932.431} C_VEL
LIN {X 0,Y 517.771,Z 488.195,A -85,B 0,C 180,E1 -4934.658,E2 -4934.658} C_VEL
LIN {X 0,Y 519.096,Z 498.922,A -85,B 0,C 180,E1 -4934.864,E2 -4934.864} C_VEL
LIN {X 0,Y 518.644,Z 597.947,A -85,B 0,C 180,E1 -4936.257,E2 -4936.257} C_VEL
LIN {X 0,Y 518.457,Z 611.443,A -85,B 0,C 180,E1 -4936.602,E2 -4936.602} C_VEL
LIN {X 0,Y 518.143,Z 624.573,A -85,B 0,C 180,E1 -4937.117,E2 -4937.117} C_VEL
LIN {X 0,Y 517.872,Z 637.164,A -85,B 0,C 180,E1 -4937.792,E2 -4937.792} C_VEL
LIN {X 0,Y 517.583,Z 648.003,A -85,B 0,C 180,E1 -4938.546,E2 -4938.546} C_VEL
LIN {X 0,Y 517.216,Z 659.272,A -85,B 0,C 180,E1 -4939.529,E2 -4939.529} C_VEL
LIN {X 0,Y 516.978,Z 667.519,A -85,B 0,C 180,E1 -4940.414,E2 -4940.414} C_VEL
LIN {X 0,Y 516.737,Z 676.477,A -85,B 0,C 180,E1 -4941.593,E2 -4941.593} C_VEL
LIN {X 0,Y 516.55,Z 683.671,A -85,B 0,C 180,E1 -4942.77,E2 -4942.77} C_VEL
LIN {X 0,Y 516.449,Z 688.558,A -85,B 0,C 180,E1 -4943.75,E2 -4943.75} C_VEL
LIN {X 0,Y 516.313,Z 693.288,A -85,B 0,C 180,E1 -4944.924,E2 -4944.924} C_VEL
LIN {X 0,Y 516.373,Z 696.908,A -85,B 0,C 180,E1 -4946.098,E2 -4946.098} C_VEL
LIN {X 0,Y 516.282,Z 698.78,A -85,B 0,C 180,E1 -4946.879,E2 -4946.879} C_VEL
LIN {X 0,Y 516.261,Z 700.21,A -85,B 0,C 180,E1 -4947.659,E2 -4947.659} C_VEL
LIN {X 0,Y 516.16,Z 701.83,A -85,B 0,C 180,E1 -4949.22,E2 -4949.22} C_VEL
LIN {X 0,Y 516.155,Z 702.067,A -85,B 0,C 180,E1 -4950,E2 -4950} C_VEL
LIN {X 0,Y 516.16,Z 701.883,A -85,B 0,C 180,E1 -4950.78,E2 -4950.78} C_VEL
LIN {X 0,Y 516.262,Z 700.336,A -85,B 0,C 180,E1 -4952.341,E2 -4952.341} C_VEL
LIN {X 0,Y 516.283,Z 698.967,A -85,B 0,C 180,E1 -4953.121,E2 -4953.121} C_VEL
LIN {X 0,Y 516.361,Z 696.102,A -85,B 0,C 180,E1 -4954.293,E2 -4954.293} C_VEL
LIN {X 0,Y 516.4,Z 692.21,A -85,B 0,C 180,E1 -4955.467,E2 -4955.467} C_VEL
LIN {X 0,Y 516.472,Z 686.4,A -85,B 0,C 180,E1 -4956.795,E2 -4956.795} C_VEL
LIN {X 0,Y 516.643,Z 679.61,A -85,B 0,C 180,E1 -4958.015,E2 -4958.015} C_VEL
LIN {X 0,Y 516.852,Z 671.443,A -85,B 0,C 180,E1 -4959.194,E2 -4959.194} C_VEL
LIN {X 0,Y 517.084,Z 663.036,A -85,B 0,C 180,E1 -4960.177,E2 -4960.177} C_VEL
LIN {X 0,Y 517.468,Z 652.722,A -85,B 0,C 180,E1 -4961.159,E2 -4961.159} C_VEL
LIN {X 0,Y 517.738,Z 642.163,A -85,B 0,C 180,E1 -4961.973,E2 -4961.973} C_VEL
LIN {X 0,Y 518.019,Z 631.277,A -85,B 0,C 180,E1 -4962.637,E2 -4962.637} C_VEL
LIN {X 0,Y 518.329,Z 618.634,A -85,B 0,C 180,E1 -4963.227,E2 -4963.227} C_VEL
LIN {X 0,Y 518.546,Z 606.14,A -85,B 0,C 180,E1 -4963.646,E2 -4963.646} C_VEL
LIN {X 0,Y 518.717,Z 593.13,A -85,B 0,C 180,E1 -4963.916,E2 -4963.916} C_VEL
LIN {X 0,Y 519.045,Z 497.549,A -85,B 0,C 180,E1 -4965.247,E2 -4965.247} C_VEL
LIN {X 0,Y 517.76,Z 488.046,A -85,B 0,C 180,E1 -4965.443,E2 -4965.443} C_VEL
LIN {X 0,Y 518.171,Z 463.766,A -85,B 0,C 180,E1 -4968.361,E2 -4968.361} C_VEL
LIN {X 0,Y 518.752,Z 438.401,A -85,B 0,C 180,E1 -4971.457,E2 -4971.457} C_VEL
LIN {X 0,Y 519.249,Z 418.209,A -85,B 0,C 180,E1 -4973.957,E2 -4973.957} C_VEL
LIN {X 0,Y 519.747,Z 397.75,A -85,B 0,C 180,E1 -4976.502,E2 -4976.502} C_VEL
LIN {X 0,Y 517.839,Z 388.265,A -85,B 0,C 180,E1 -4977.759,E2 -4977.759} C_VEL
LIN {X 0,Y 516.904,Z 384.199,A -85,B 0,C 180,E1 -4978.342,E2 -4978.342} C_VEL
LIN {X 0,Y 516.89,Z 384.101,A -85,B 0,C 180,E1 -4981.11,E2 -4981.11} C_VEL
LIN {X 0,Y 516.895,Z 384.098,A -85,B 0,C 180,E1 -4983.963,E2 -4983.963} C_VEL
LIN {X 0,Y 516.818,Z 384.101,A -85,B 0,C 180,E1 -4986.751,E2 -4986.751} C_VEL
LIN {X 0,Y 516.863,Z 384.099,A -85,B 0,C 180,E1 -4989.724,E2 -4989.724} C_VEL
LIN {X 0,Y 516.844,Z 384.101,A -85,B 0,C 180,E1 -4992.836,E2 -4992.836} C_VEL
LIN {X 0,Y 516.899,Z 384.087,A -85,B 0,C 180,E1 -4995.007,E2 -4995.007} C_VEL
LIN {X 0,Y 516.889,Z 384.095,A -85,B 0,C 180,E1 -4998.402,E2 -4998.402} C_VEL
LIN {X 0,Y 516.877,Z 384.1,A -85,B 0,C 180,E1 -5001.283,E2 -5001.283} C_VEL
LIN {X 0,Y 516.857,Z 384.099,A -85,B 0,C 180,E1 -5004.673,E2 -5004.673} C_VEL
LIN {X 0,Y 516.898,Z 384.095,A -85,B 0,C 180,E1 -5007.457,E2 -5007.457} C_VEL
LIN {X 0,Y 516.906,Z 384.089,A -85,B 0,C 180,E1 -5010.694,E2 -5010.694} C_VEL
LIN {X 0,Y 516.882,Z 384.103,A -85,B 0,C 180,E1 -5013.819,E2 -5013.819} C_VEL
LIN {X 0,Y 516.861,Z 384.093,A -85,B 0,C 180,E1 -5016.776,E2 -5016.776} C_VEL
LIN {X 0,Y 516.933,Z 384.097,A -85,B 0,C 180,E1 -5019.735,E2 -5019.735} C_VEL
LIN {X 0,Y 516.883,Z 384.09,A -85,B 0,C 180,E1 -5022.594,E2 -5022.594} C_VEL
LIN {X 0,Y 516.94,Z 384.089,A -85,B 0,C 180,E1 -5025.03,E2 -5025.03} C_VEL
LIN {X 0,Y 516.93,Z 384.084,A -85,B 0,C 180,E1 -5028.233,E2 -5028.233} C_VEL
LIN {X 0,Y 516.93,Z 384.092,A -85,B 0,C 180,E1 -5031.399,E2 -5031.399} C_VEL
LIN {X 0,Y 516.986,Z 384.077,A -85,B 0,C 180,E1 -5034.539,E2 -5034.539} C_VEL
LIN {X 0,Y 517.076,Z 384.075,A -85,B 0,C 180,E1 -5037.663,E2 -5037.663} C_VEL
LIN {X 0,Y 517.069,Z 384.075,A -85,B 0,C 180,E1 -5040,E2 -5040} C_VEL
LIN {X 0,Y 517.076,Z 384.065,A -85,B 0,C 180,E1 -5042.337,E2 -5042.337} C_VEL
LIN {X 0,Y 516.971,Z 384.086,A -85,B 0,C 180,E1 -5046.244,E2 -5046.244} C_VEL
LIN {X 0,Y 516.91,Z 384.09,A -85,B 0,C 180,E1 -5049.39,E2 -5049.39} C_VEL
LIN {X 0,Y 516.902,Z 384.093,A -85,B 0,C 180,E1 -5052.565,E2 -5052.565} C_VEL
LIN {X 0,Y 516.832,Z 384.103,A -85,B 0,C 180,E1 -5055.781,E2 -5055.781} C_VEL
LIN {X 0,Y 516.85,Z 384.102,A -85,B 0,C 180,E1 -5058.225,E2 -5058.225} C_VEL
LIN {X 0,Y 516.87,Z 384.096,A -85,B 0,C 180,E1 -5060.703,E2 -5060.703} C_VEL
LIN {X 0,Y 516.859,Z 384.093,A -85,B 0,C 180,E1 -5063.224,E2 -5063.224} C_VEL
LIN {X 0,Y 516.863,Z 384.101,A -85,B 0,C 180,E1 -5066.177,E2 -5066.177} C_VEL
LIN {X 0,Y 516.906,Z 384.089,A -85,B 0,C 180,E1 -5069.306,E2 -5069.306} C_VEL
LIN {X 0,Y 516.852,Z 384.105,A -85,B 0,C 180,E1 -5072.027,E2 -5072.027} C_VEL
LIN {X 0,Y 516.872,Z 384.093,A -85,B 0,C 180,E1 -5074.826,E2 -5074.826} C_VEL
LIN {X 0,Y 516.854,Z 384.104,A -85,B 0,C 180,E1 -5077.939,E2 -5077.939} C_VEL
LIN {X 0,Y 516.821,Z 384.089,A -85,B 0,C 180,E1 -5080.748,E2 -5080.748} C_VEL
LIN {X 0,Y 516.862,Z 384.101,A -85,B 0,C 180,E1 -5083.906,E2 -5083.906} C_VEL
LIN {X 0,Y 516.862,Z 384.101,A -85,B 0,C 180,E1 -5086.11,E2 -5086.11} C_VEL
LIN {X 0,Y 516.821,Z 384.09,A -85,B 0,C 180,E1 -5089.252,E2 -5089.252} C_VEL
LIN {X 0,Y 516.853,Z 384.106,A -85,B 0,C 180,E1 -5092.061,E2 -5092.061} C_VEL
LIN {X 0,Y 516.853,Z 384.101,A -85,B 0,C 180,E1 -5095.173,E2 -5095.173} C_VEL
LIN {X 0,Y 516.847,Z 384.108,A -85,B 0,C 180,E1 -5097.973,E2 -5097.973} C_VEL
LIN {X 0,Y 516.892,Z 384.285,A -85,B 0,C 180,E1 -5101.056,E2 -5101.056} C_VEL
LIN {X 0,Y 519.719,Z 396.826,A -85,B 0,C 180,E1 -5102.805,E2 -5102.805} C_VEL
LIN {X 0,Y 519.735,Z 405.881,A -85,B 0,C 180,E1 -5103.929,E2 -5103.929} C_VEL
LIN {X 0,Y 518.956,Z 431.497,A -85,B 0,C 180,E1 -5107.058,E2 -5107.058} C_VEL
LIN {X 0,Y 518.377,Z 452.293,A -85,B 0,C 180,E1 -5109.567,E2 -5109.567} C_VEL
LIN {X 0,Y 517.852,Z 480.103,A -85,B 0,C 180,E1 -5112.832,E2 -5112.832} C_VEL
LIN {X 0,Y 517.566,Z 495.272,A -85,B 0,C 180,E1 -5114.603,E2 -5114.603} C_VEL
LIN {X 0,Y 519.038,Z 508.587,A -85,B 0,C 180,E1 -5114.856,E2 -5114.856} C_VEL
LIN {X 0,Y 518.513,Z 605.551,A -85,B 0,C 180,E1 -5116.254,E2 -5116.254} C_VEL
LIN {X 0,Y 518.254,Z 618.843,A -85,B 0,C 180,E1 -5116.596,E2 -5116.596} C_VEL
LIN {X 0,Y 517.996,Z 632.233,A -85,B 0,C 180,E1 -5117.113,E2 -5117.113} C_VEL
LIN {X 0,Y 517.706,Z 645.088,A -85,B 0,C 180,E1 -5117.802,E2 -5117.802} C_VEL
LIN {X 0,Y 517.375,Z 657.219,A -85,B 0,C 180,E1 -5118.64,E2 -5118.64} C_VEL
LIN {X 0,Y 517.06,Z 667.396,A -85,B 0,C 180,E1 -5119.525,E2 -5119.525} C_VEL
LIN {X 0,Y 516.824,Z 677.487,A -85,B 0,C 180,E1 -5120.608,E2 -5120.608} C_VEL
LIN {X 0,Y 516.644,Z 686.337,A -85,B 0,C 180,E1 -5121.788,E2 -5121.788} C_VEL
LIN {X 0,Y 516.507,Z 693.43,A -85,B 0,C 180,E1 -5122.966,E2 -5122.966} C_VEL
LIN {X 0,Y 516.456,Z 699.107,A -85,B 0,C 180,E1 -5124.142,E2 -5124.142} C_VEL
LIN {X 0,Y 516.324,Z 703.546,A -85,B 0,C 180,E1 -5125.315,E2 -5125.315} C_VEL
LIN {X 0,Y 516.403,Z 705.912,A -85,B 0,C 180,E1 -5126.098,E2 -5126.098} C_VEL
LIN {X 0,Y 516.315,Z 707.807,A -85,B 0,C 180,E1 -5126.879,E2 -5126.879} C_VEL
LIN {X 0,Y 516.282,Z 709.245,A -85,B 0,C 180,E1 -5127.659,E2 -5127.659} C_VEL
LIN {X 0,Y 516.226,Z 710.257,A -85,B 0,C 180,E1 -5128.44,E2 -5128.44} C_VEL
LIN {X 0,Y 516.203,Z 710.872,A -85,B 0,C 180,E1 -5129.22,E2 -5129.22} C_VEL
LIN {X 0,Y 516.201,Z 711.088,A -85,B 0,C 180,E1 -5130,E2 -5130} C_VEL
LIN {X 0,Y 516.204,Z 710.862,A -85,B 0,C 180,E1 -5130.78,E2 -5130.78} C_VEL
LIN {X 0,Y 516.229,Z 710.238,A -85,B 0,C 180,E1 -5131.56,E2 -5131.56} C_VEL
LIN {X 0,Y 516.286,Z 709.213,A -85,B 0,C 180,E1 -5132.34,E2 -5132.34} C_VEL
LIN {X 0,Y 516.32,Z 707.768,A -85,B 0,C 180,E1 -5133.121,E2 -5133.121} C_VEL
LIN {X 0,Y 516.365,Z 704.733,A -85,B 0,C 180,E1 -5134.293,E2 -5134.293} C_VEL
LIN {X 0,Y 516.411,Z 700.623,A -85,B 0,C 180,E1 -5135.467,E2 -5135.467} C_VEL
LIN {X 0,Y 516.495,Z 694.397,A -85,B 0,C 180,E1 -5136.821,E2 -5136.821} C_VEL
LIN {X 0,Y 516.629,Z 687.395,A -85,B 0,C 180,E1 -5138.015,E2 -5138.015} C_VEL
LIN {X 0,Y 516.792,Z 678.813,A -85,B 0,C 180,E1 -5139.195,E2 -5139.195} C_VEL
LIN {X 0,Y 517.061,Z 668.998,A -85,B 0,C 180,E1 -5140.276,E2 -5140.276} C_VEL
LIN {X 0,Y 517.322,Z 657.92,A -85,B 0,C 180,E1 -5141.262,E2 -5141.262} C_VEL
LIN {X 0,Y 517.612,Z 646.06,A -85,B 0,C 180,E1 -5142.098,E2 -5142.098} C_VEL
LIN {X 0,Y 517.873,Z 633.416,A -85,B 0,C 180,E1 -5142.79,E2 -5142.79} C_VEL
LIN {X 0,Y 518.189,Z 620.76,A -85,B 0,C 180,E1 -5143.305,E2 -5143.305} C_VEL
LIN {X 0,Y 518.412,Z 607.465,A -85,B 0,C 180,E1 -5143.674,E2 -5143.674} C_VEL
LIN {X 0,Y 518.6,Z 583.85,A -85,B 0,C 180,E1 -5144.044,E2 -5144.044} C_VEL
LIN {X 0,Y 518.782,Z 506.191,A -85,B 0,C 180,E1 -5145.157,E2 -5145.157} C_VEL
LIN {X 0,Y 517.481,Z 493.813,A -85,B 0,C 180,E1 -5145.399,E2 -5145.399} C_VEL
LIN {X 0,Y 517.887,Z 467.884,A -85,B 0,C 180,E1 -5148.371,E2 -5148.371} C_VEL
LIN {X 0,Y 518.355,Z 441.21,A -85,B 0,C 180,E1 -5151.474,E2 -5151.474} C_VEL
LIN {X 0,Y 518.948,Z 414.794,A -85,B 0,C 180,E1 -5154.61,E2 -5154.61} C_VEL
LIN {X 0,Y 519.326,Z 396.84,A -85,B 0,C 180,E1 -5156.802,E2 -5156.802} C_VEL
LIN {X 0,Y 517.445,Z 386.856,A -85,B 0,C 180,E1 -5158.146,E2 -5158.146} C_VEL
LIN {X 0,Y 516.87,Z 384.204,A -85,B 0,C 180,E1 -5158.557,E2 -5158.557} C_VEL
LIN {X 0,Y 516.849,Z 384.104,A -85,B 0,C 180,E1 -5161.112,E2 -5161.112} C_VEL
LIN {X 0,Y 516.87,Z 384.106,A -85,B 0,C 180,E1 -5163.959,E2 -5163.959} C_VEL
LIN {X 0,Y 516.808,Z 384.107,A -85,B 0,C 180,E1 -5166.752,E2 -5166.752} C_VEL
LIN {X 0,Y 516.86,Z 384.101,A -85,B 0,C 180,E1 -5169.19,E2 -5169.19} C_VEL
LIN {X 0,Y 516.833,Z 384.109,A -85,B 0,C 180,E1 -5171.783,E2 -5171.783} C_VEL
LIN {X 0,Y 516.897,Z 384.095,A -85,B 0,C 180,E1 -5175.007,E2 -5175.007} C_VEL
LIN {X 0,Y 516.855,Z 384.1,A -85,B 0,C 180,E1 -5178.406,E2 -5178.406} C_VEL
LIN {X 0,Y 516.875,Z 384.101,A -85,B 0,C 180,E1 -5181.283,E2 -5181.283} C_VEL
LIN {X 0,Y 516.863,Z 384.099,A -85,B 0,C 180,E1 -5184.671,E2 -5184.671} C_VEL
LIN {X 0,Y 516.897,Z 384.1,A -85,B 0,C 180,E1 -5187.457,E2 -5187.457} C_VEL
LIN {X 0,Y 516.923,Z 384.092,A -85,B 0,C 180,E1 -5190.695,E2 -5190.695} C_VEL
LIN {X 0,Y 516.898,Z 384.098,A -85,B 0,C 180,E1 -5193.815,E2 -5193.815} C_VEL
LIN {X 0,Y 516.862,Z 384.101,A -85,B 0,C 180,E1 -5196.776,E2 -5196.776} C_VEL
LIN {X 0,Y 516.943,Z 384.094,A -85,B 0,C 180,E1 -5199.732,E2 -5199.732} C_VEL
LIN {X 0,Y 516.91,Z 384.097,A -85,B 0,C 180,E1 -5202.595,E2 -5202.595} C_VEL
LIN {X 0,Y 517,Z 384.286,A -85,B 0,C 180,E1 -5205.032,E2 -5205.032} C_VEL
LIN {X 0,Y 517.18,Z 385.236,A -85,B 0,C 180,E1 -5205.151,E2 -5205.151} C_VEL
LIN {X 0,Y 518.827,Z 390.139,A -85,B 0,C 180,E1 -5205.294,E2 -5205.294} C_VEL
LIN {X 0,Y 518.562,Z 466.528,A -85,B 0,C 180,E1 -5206.455,E2 -5206.455} C_VEL
LIN {X 0,Y 518.457,Z 479.239,A -85,B 0,C 180,E1 -5206.801,E2 -5206.801} C_VEL
LIN {X 0,Y 518.33,Z 492.15,A -85,B 0,C 180,E1 -5207.321,E2 -5207.321} C_VEL
LIN {X 0,Y 518.12,Z 504.501,A -85,B 0,C 180,E1 -5208.005,E2 -5208.005} C_VEL
LIN {X 0,Y 517.947,Z 515.048,A -85,B 0,C 180,E1 -5208.752,E2 -5208.752} C_VEL
LIN {X 0,Y 517.658,Z 525.115,A -85,B 0,C 180,E1 -5209.637,E2 -5209.637} C_VEL
LIN {X 0,Y 517.468,Z 534.108,A -85,B 0,C 180,E1 -5210.62,E2 -5210.62} C_VEL
LIN {X 0,Y 517.191,Z 542.837,A -85,B 0,C 180,E1 -5211.797,E2 -5211.797} C_VEL
LIN {X 0,Y 516.97,Z 549.806,A -85,B 0,C 180,E1 -5212.972,E2 -5212.972} C_VEL
LIN {X 0,Y 516.911,Z 555.302,A -85,B 0,C 180,E1 -5214.147,E2 -5214.147} C_VEL
LIN {X 0,Y 516.735,Z 559.619,A -85,B 0,C 180,E1 -5215.319,E2 -5215.319} C_VEL
LIN {X 0,Y 516.683,Z 561.878,A -85,B 0,C 180,E1 -5216.1,E2 -5216.1} C_VEL
LIN {X 0,Y 516.704,Z 563.704,A -85,B 0,C 180,E1 -5216.881,E2 -5216.881} C_VEL
LIN {X 0,Y 516.598,Z 565.111,A -85,B 0,C 180,E1 -5217.661,E2 -5217.661} C_VEL
LIN {X 0,Y 516.615,Z 566.07,A -85,B 0,C 180,E1 -5218.441,E2 -5218.441} C_VEL
LIN {X 0,Y 516.555,Z 566.859,A -85,B 0,C 180,E1 -5220,E2 -5220} C_VEL
LIN {X 0,Y 516.568,Z 566.64,A -85,B 0,C 180,E1 -5220.78,E2 -5220.78} C_VEL
LIN {X 0,Y 516.589,Z 565.018,A -85,B 0,C 180,E1 -5222.339,E2 -5222.339} C_VEL
LIN {X 0,Y 516.593,Z 563.626,A -85,B 0,C 180,E1 -5223.12,E2 -5223.12} C_VEL
LIN {X 0,Y 516.709,Z 560.696,A -85,B 0,C 180,E1 -5224.29,E2 -5224.29} C_VEL
LIN {X 0,Y 516.732,Z 556.753,A -85,B 0,C 180,E1 -5225.463,E2 -5225.463} C_VEL
LIN {X 0,Y 516.897,Z 551.421,A -85,B 0,C 180,E1 -5226.683,E2 -5226.683} C_VEL
LIN {X 0,Y 517.042,Z 545.213,A -85,B 0,C 180,E1 -5227.812,E2 -5227.812} C_VEL
LIN {X 0,Y 517.275,Z 537.178,A -85,B 0,C 180,E1 -5228.989,E2 -5228.989} C_VEL
LIN {X 0,Y 517.423,Z 528.966,A -85,B 0,C 180,E1 -5229.973,E2 -5229.973} C_VEL
LIN {X 0,Y 517.665,Z 518.876,A -85,B 0,C 180,E1 -5230.957,E2 -5230.957} C_VEL
LIN {X 0,Y 517.994,Z 508.828,A -85,B 0,C 180,E1 -5231.743,E2 -5231.743} C_VEL
LIN {X 0,Y 518.167,Z 497.453,A -85,B 0,C 180,E1 -5232.459,E2 -5232.459} C_VEL
LIN {X 0,Y 518.344,Z 485.762,A -85,B 0,C 180,E1 -5233.027,E2 -5233.027} C_VEL
LIN {X 0,Y 518.539,Z 473.129,A -85,B 0,C 180,E1 -5233.471,E2 -5233.471} C_VEL
LIN {X 0,Y 518.604,Z 459.939,A -85,B 0,C 180,E1 -5233.769,E2 -5233.769} C_VEL
LIN {X 0,Y 518.866,Z 390.183,A -85,B 0,C 180,E1 -5234.794,E2 -5234.794} C_VEL
LIN {X 0,Y 517.135,Z 384.897,A -85,B 0,C 180,E1 -5234.952,E2 -5234.952} C_VEL
LIN {X 0,Y 516.962,Z 384.149,A -85,B 0,C 180,E1 -5235.11,E2 -5235.11} C_VEL
LIN {X 0,Y 516.92,Z 384.096,A -85,B 0,C 180,E1 -5238.223,E2 -5238.223} C_VEL
LIN {X 0,Y 516.916,Z 384.1,A -85,B 0,C 180,E1 -5240.701,E2 -5240.701} C_VEL
LIN {X 0,Y 516.906,Z 384.094,A -85,B 0,C 180,E1 -5244.072,E2 -5244.072} C_VEL
LIN {X 0,Y 516.901,Z 384.101,A -85,B 0,C 180,E1 -5246.659,E2 -5246.659} C_VEL
LIN {X 0,Y 516.913,Z 384.089,A -85,B 0,C 180,E1 -5249.524,E2 -5249.524} C_VEL
LIN {X 0,Y 516.897,Z 384.1,A -85,B 0,C 180,E1 -5252.543,E2 -5252.543} C_VEL
LIN {X 0,Y 516.866,Z 384.099,A -85,B 0,C 180,E1 -5255.329,E2 -5255.329} C_VEL
LIN {X 0,Y 516.881,Z 384.094,A -85,B 0,C 180,E1 -5257.943,E2 -5257.943} C_VEL
LIN {X 0,Y 516.881,Z 384.096,A -85,B 0,C 180,E1 -5259.422,E2 -5259.422} C_VEL
LIN {X 0,Y 516.213,Z 384.182,A -85,B 0,C 180,E1 -5260.072,E2 -5260.072} C_VEL
LIN {X 0,Y 513.347,Z 384.537,A -85,B 0,C 180,E1 -5261.129,E2 -5261.129} C_VEL
LIN {X 0,Y 510.924,Z 384.84,A -85,B 0,C 180,E1 -5261.98,E2 -5261.98} C_VEL
LIN {X 0,Y 509.885,Z 384.972,A -85,B 0,C 180,E1 -5262.637,E2 -5262.637} C_VEL
LIN {X 0,Y 509.802,Z 384.981,A -85,B 0,C 180,E1 -5262.859,E2 -5262.859} C_VEL
LIN {X 0,Y 509.824,Z 384.974,A -85,B 0,C 180,E1 -5265.793,E2 -5265.793} C_VEL
LIN {X 0,Y 509.855,Z 384.977,A -85,B 0,C 180,E1 -5268.574,E2 -5268.574} C_VEL
LIN {X 0,Y 509.852,Z 384.965,A -85,B 0,C 180,E1 -5271.787,E2 -5271.787} C_VEL
LIN {X 0,Y 509.83,Z 384.975,A -85,B 0,C 180,E1 -5274.622,E2 -5274.622} C_VEL
LIN {X 0,Y 509.864,Z 384.968,A -85,B 0,C 180,E1 -5277.481,E2 -5277.481} C_VEL
LIN {X 0,Y 509.861,Z 384.974,A -85,B 0,C 180,E1 -5280.274,E2 -5280.274} C_VEL
LIN {X 0,Y 509.927,Z 385.22,A -85,B 0,C 180,E1 -5281.569,E2 -5281.569} C_VEL
LIN {X 0,Y 512.898,Z 398.663,A -85,B 0,C 180,E1 -5283.402,E2 -5283.402} C_VEL
LIN {X 0,Y 512.29,Z 423.791,A -85,B 0,C 180,E1 -5286.556,E2 -5286.556} C_VEL
LIN {X 0,Y 511.667,Z 445.649,A -85,B 0,C 180,E1 -5289.287,E2 -5289.287} C_VEL
LIN {X 0,Y 511.101,Z 469.296,A -85,B 0,C 180,E1 -5292.189,E2 -5292.189} C_VEL
LIN {X 0,Y 510.809,Z 488.069,A -85,B 0,C 180,E1 -5294.44,E2 -5294.44} C_VEL
LIN {X 0,Y 512.245,Z 498.546,A -85,B 0,C 180,E1 -5294.652,E2 -5294.652} C_VEL
LIN {X 0,Y 511.755,Z 597.904,A -85,B 0,C 180,E1 -5296.069,E2 -5296.069} C_VEL
LIN {X 0,Y 511.55,Z 611.446,A -85,B 0,C 180,E1 -5296.418,E2 -5296.418} C_VEL
LIN {X 0,Y 511.212,Z 624.598,A -85,B 0,C 180,E1 -5296.94,E2 -5296.94} C_VEL
LIN {X 0,Y 510.928,Z 636.654,A -85,B 0,C 180,E1 -5297.59,E2 -5297.59} C_VEL
LIN {X 0,Y 510.615,Z 648.046,A -85,B 0,C 180,E1 -5298.387,E2 -5298.387} C_VEL
LIN {X 0,Y 510.23,Z 659.319,A -85,B 0,C 180,E1 -5299.384,E2 -5299.384} C_VEL
LIN {X 0,Y 509.97,Z 667.569,A -85,B 0,C 180,E1 -5300.281,E2 -5300.281} C_VEL
LIN {X 0,Y 509.707,Z 676.529,A -85,B 0,C 180,E1 -5301.476,E2 -5301.476} C_VEL
LIN {X 0,Y 509.488,Z 683.725,A -85,B 0,C 180,E1 -5302.669,E2 -5302.669} C_VEL
LIN {X 0,Y 509.387,Z 688.611,A -85,B 0,C 180,E1 -5303.663,E2 -5303.663} C_VEL
LIN {X 0,Y 509.248,Z 693.342,A -85,B 0,C 180,E1 -5304.853,E2 -5304.853} C_VEL
LIN {X 0,Y 509.285,Z 696.965,A -85,B 0,C 180,E1 -5306.044,E2 -5306.044} C_VEL
LIN {X 0,Y 509.201,Z 698.832,A -85,B 0,C 180,E1 -5306.835,E2 -5306.835} C_VEL
LIN {X 0,Y 509.19,Z 700.262,A -85,B 0,C 180,E1 -5307.627,E2 -5307.627} C_VEL
LIN {X 0,Y 509.074,Z 701.882,A -85,B 0,C 180,E1 -5309.209,E2 -5309.209} C_VEL
LIN {X 0,Y 509.066,Z 702.121,A -85,B 0,C 180,E1 -5310,E2 -5310} C_VEL
LIN {X 0,Y 509.073,Z 701.935,A -85,B 0,C 180,E1 -5310.791,E2 -5310.791} C_VEL
LIN {X 0,Y 509.19,Z 700.385,A -85,B 0,C 180,E1 -5312.373,E2 -5312.373} C_VEL
LIN {X 0,Y 509.202,Z 699.024,A -85,B 0,C 180,E1 -5313.165,E2 -5313.165} C_VEL
LIN {X 0,Y 509.265,Z 696.156,A -85,B 0,C 180,E1 -5314.353,E2 -5314.353} C_VEL
LIN {X 0,Y 509.338,Z 692.259,A -85,B 0,C 180,E1 -5315.543,E2 -5315.543} C_VEL
LIN {X 0,Y 509.382,Z 687.216,A -85,B 0,C 180,E1 -5316.735,E2 -5316.735} C_VEL
LIN {X 0,Y 509.566,Z 680.854,A -85,B 0,C 180,E1 -5317.928,E2 -5317.928} C_VEL
LIN {X 0,Y 509.77,Z 672.956,A -85,B 0,C 180,E1 -5319.123,E2 -5319.123} C_VEL
LIN {X 0,Y 510.03,Z 664.895,A -85,B 0,C 180,E1 -5320.119,E2 -5320.119} C_VEL
LIN {X 0,Y 510.385,Z 655.013,A -85,B 0,C 180,E1 -5321.115,E2 -5321.115} C_VEL
LIN {X 0,Y 510.75,Z 643.645,A -85,B 0,C 180,E1 -5322.033,E2 -5322.033} C_VEL
LIN {X 0,Y 511.035,Z 633.091,A -85,B 0,C 180,E1 -5322.712,E2 -5322.712} C_VEL
LIN {X 0,Y 511.349,Z 621.034,A -85,B 0,C 180,E1 -5323.31,E2 -5323.31} C_VEL
LIN {X 0,Y 511.599,Z 607.79,A -85,B 0,C 180,E1 -5323.784,E2 -5323.784} C_VEL
LIN {X 0,Y 511.834,Z 594.587,A -85,B 0,C 180,E1 -5324.081,E2 -5324.081} C_VEL
LIN {X 0,Y 512.157,Z 497.526,A -85,B 0,C 180,E1 -5325.455,E2 -5325.455} C_VEL
LIN {X 0,Y 510.798,Z 487.942,A -85,B 0,C 180,E1 -5325.662,E2 -5325.662} C_VEL
LIN {X 0,Y 511.221,Z 463.469,A -85,B 0,C 180,E1 -5328.62,E2 -5328.62} C_VEL
LIN {X 0,Y 511.893,Z 437.992,A -85,B 0,C 180,E1 -5331.759,E2 -5331.759} C_VEL
LIN {X 0,Y 512.472,Z 416.068,A -85,B 0,C 180,E1 -5334.51,E2 -5334.51} C_VEL
LIN {X 0,Y 512.889,Z 398.906,A -85,B 0,C 180,E1 -5336.665,E2 -5336.665} C_VEL
LIN {X 0,Y 509.873,Z 385.105,A -85,B 0,C 180,E1 -5338.558,E2 -5338.558} C_VEL
LIN {X 0,Y 509.821,Z 384.979,A -85,B 0,C 180,E1 -5341.59,E2 -5341.59} C_VEL
LIN {X 0,Y 509.841,Z 384.975,A -85,B 0,C 180,E1 -5344.415,E2 -5344.415} C_VEL
LIN {X 0,Y 509.786,Z 384.981,A -85,B 0,C 180,E1 -5347.344,E2 -5347.344} C_VEL
LIN {X 0,Y 509.816,Z 384.972,A -85,B 0,C 180,E1 -5350.385,E2 -5350.385} C_VEL
LIN {X 0,Y 509.808,Z 384.98,A -85,B 0,C 180,E1 -5353.574,E2 -5353.574} C_VEL
LIN {X 0,Y 509.811,Z 384.977,A -85,B 0,C 180,E1 -5356.427,E2 -5356.427} C_VEL
LIN {X 0,Y 509.815,Z 384.98,A -85,B 0,C 180,E1 -5359.306,E2 -5359.306} C_VEL
LIN {X 0,Y 509.819,Z 384.979,A -85,B 0,C 180,E1 -5361.792,E2 -5361.792} C_VEL
LIN {X 0,Y 509.821,Z 384.975,A -85,B 0,C 180,E1 -5364.621,E2 -5364.621} C_VEL
LIN {X 0,Y 509.864,Z 384.971,A -85,B 0,C 180,E1 -5367.481,E2 -5367.481} C_VEL
LIN {X 0,Y 509.856,Z 384.969,A -85,B 0,C 180,E1 -5370.275,E2 -5370.275} C_VEL
LIN {X 0,Y 509.822,Z 384.975,A -85,B 0,C 180,E1 -5372.941,E2 -5372.941} C_VEL
LIN {X 0,Y 509.839,Z 384.978,A -85,B 0,C 180,E1 -5375.572,E2 -5375.572} C_VEL
LIN {X 0,Y 509.824,Z 384.978,A -85,B 0,C 180,E1 -5378.149,E2 -5378.149} C_VEL
LIN {X 0,Y 509.851,Z 384.969,A -85,B 0,C 180,E1 -5380.681,E2 -5380.681} C_VEL
LIN {X 0,Y 509.801,Z 384.974,A -85,B 0,C 180,E1 -5383.172,E2 -5383.172} C_VEL
LIN {X 0,Y 509.857,Z 384.978,A -85,B 0,C 180,E1 -5385.634,E2 -5385.634} C_VEL
LIN {X 0,Y 509.894,Z 384.961,A -85,B 0,C 180,E1 -5388.131,E2 -5388.131} C_VEL
LIN {X 0,Y 509.882,Z 384.969,A -85,B 0,C 180,E1 -5391.279,E2 -5391.279} C_VEL
LIN {X 0,Y 509.923,Z 384.967,A -85,B 0,C 180,E1 -5393.67,E2 -5393.67} C_VEL
LIN {X 0,Y 509.887,Z 384.963,A -85,B 0,C 180,E1 -5396.839,E2 -5396.839} C_VEL
LIN {X 0,Y 509.925,Z 384.963,A -85,B 0,C 180,E1 -5398.42,E2 -5398.42} C_VEL
LIN {X 0,Y 510.037,Z 384.951,A -85,B 0,C 180,E1 -5400,E2 -5400} C_VEL
LIN {X 0,Y 510.044,Z 384.94,A -85,B 0,C 180,E1 -5402.369,E2 -5402.369} C_VEL
LIN {X 0,Y 509.938,Z 384.964,A -85,B 0,C 180,E1 -5405.536,E2 -5405.536} C_VEL
LIN {X 0,Y 509.878,Z 384.969,A -85,B 0,C 180,E1 -5407.923,E2 -5407.923} C_VEL
LIN {X 0,Y 509.865,Z 384.966,A -85,B 0,C 180,E1 -5411.127,E2 -5411.127} C_VEL
LIN {X 0,Y 509.826,Z 384.979,A -85,B 0,C 180,E1 -5413.553,E2 -5413.553} C_VEL
LIN {X 0,Y 509.792,Z 384.976,A -85,B 0,C 180,E1 -5416.005,E2 -5416.005} C_VEL
LIN {X 0,Y 509.812,Z 384.976,A -85,B 0,C 180,E1 -5418.486,E2 -5418.486} C_VEL
LIN {X 0,Y 509.821,Z 384.974,A -85,B 0,C 180,E1 -5421.003,E2 -5421.003} C_VEL
LIN {X 0,Y 509.815,Z 384.974,A -85,B 0,C 180,E1 -5423.564,E2 -5423.564} C_VEL
LIN {X 0,Y 509.803,Z 384.979,A -85,B 0,C 180,E1 -5426.353,E2 -5426.353} C_VEL
LIN {X 0,Y 509.836,Z 384.967,A -85,B 0,C 180,E1 -5428.847,E2 -5428.847} C_VEL
LIN {X 0,Y 509.806,Z 384.981,A -85,B 0,C 180,E1 -5431.591,E2 -5431.591} C_VEL
LIN {X 0,Y 509.835,Z 384.971,A -85,B 0,C 180,E1 -5434.415,E2 -5434.415} C_VEL
LIN {X 0,Y 509.778,Z 384.983,A -85,B 0,C 180,E1 -5437.344,E2 -5437.344} C_VEL
LIN {X 0,Y 509.788,Z 384.966,A -85,B 0,C 180,E1 -5440.387,E2 -5440.387} C_VEL
LIN {X 0,Y 509.793,Z 384.975,A -85,B 0,C 180,E1 -5443.575,E2 -5443.575} C_VEL
LIN {X 0,Y 509.794,Z 384.978,A -85,B 0,C 180,E1 -5446.425,E2 -5446.425} C_VEL
LIN {X 0,Y 509.787,Z 384.969,A -85,B 0,C 180,E1 -5449.612,E2 -5449.612} C_VEL
LIN {X 0,Y 509.776,Z 384.982,A -85,B 0,C 180,E1 -5452.655,E2 -5452.655} C_VEL
LIN {X 0,Y 509.83,Z 384.982,A -85,B 0,C 180,E1 -5455.802,E2 -5455.802} C_VEL
LIN {X 0,Y 509.816,Z 384.981,A -85,B 0,C 180,E1 -5458.726,E2 -5458.726} C_VEL
LIN {X 0,Y 509.855,Z 385.176,A -85,B 0,C 180,E1 -5460.83,E2 -5460.83} C_VEL
LIN {X 0,Y 512.79,Z 398.008,A -85,B 0,C 180,E1 -5462.638,E2 -5462.638} C_VEL
LIN {X 0,Y 512.954,Z 403.468,A -85,B 0,C 180,E1 -5463.339,E2 -5463.339} C_VEL
LIN {X 0,Y 512.172,Z 427.595,A -85,B 0,C 180,E1 -5466.336,E2 -5466.336} C_VEL
LIN {X 0,Y 511.48,Z 451.205,A -85,B 0,C 180,E1 -5469.231,E2 -5469.231} C_VEL
LIN {X 0,Y 510.852,Z 477.604,A -85,B 0,C 180,E1 -5472.382,E2 -5472.382} C_VEL
LIN {X 0,Y 510.553,Z 494.607,A -85,B 0,C 180,E1 -5474.394,E2 -5474.394} C_VEL
LIN {X 0,Y 512.122,Z 509.943,A -85,B 0,C 180,E1 -5474.683,E2 -5474.683} C_VEL
LIN {X 0,Y 511.576,Z 605.035,A -85,B 0,C 180,E1 -5476.089,E2 -5476.089} C_VEL
LIN {X 0,Y 511.277,Z 618.187,A -85,B 0,C 180,E1 -5476.435,E2 -5476.435} C_VEL
LIN {X 0,Y 511.012,Z 630.943,A -85,B 0,C 180,E1 -5476.934,E2 -5476.934} C_VEL
LIN {X 0,Y 510.749,Z 642.522,A -85,B 0,C 180,E1 -5477.545,E2 -5477.545} C_VEL
LIN {X 0,Y 510.425,Z 654.805,A -85,B 0,C 180,E1 -5478.383,E2 -5478.383} C_VEL
LIN {X 0,Y 510.106,Z 665.297,A -85,B 0,C 180,E1 -5479.281,E2 -5479.281} C_VEL
LIN {X 0,Y 509.834,Z 674.768,A -85,B 0,C 180,E1 -5480.278,E2 -5480.278} C_VEL
LIN {X 0,Y 509.619,Z 683.974,A -85,B 0,C 180,E1 -5481.474,E2 -5481.474} C_VEL
LIN {X 0,Y 509.435,Z 691.347,A -85,B 0,C 180,E1 -5482.668,E2 -5482.668} C_VEL
LIN {X 0,Y 509.39,Z 698.144,A -85,B 0,C 180,E1 -5484.06,E2 -5484.06} C_VEL
LIN {X 0,Y 509.267,Z 702.592,A -85,B 0,C 180,E1 -5485.25,E2 -5485.25} C_VEL
LIN {X 0,Y 509.357,Z 704.951,A -85,B 0,C 180,E1 -5486.044,E2 -5486.044} C_VEL
LIN {X 0,Y 509.267,Z 706.85,A -85,B 0,C 180,E1 -5486.835,E2 -5486.835} C_VEL
LIN {X 0,Y 509.235,Z 708.301,A -85,B 0,C 180,E1 -5487.627,E2 -5487.627} C_VEL
LIN {X 0,Y 509.166,Z 709.916,A -85,B 0,C 180,E1 -5489.209,E2 -5489.209} C_VEL
LIN {X 0,Y 509.188,Z 710.131,A -85,B 0,C 180,E1 -5490,E2 -5490} C_VEL
LIN {X 0,Y 509.194,Z 709.899,A -85,B 0,C 180,E1 -5490.791,E2 -5490.791} C_VEL
LIN {X 0,Y 509.246,Z 708.217,A -85,B 0,C 180,E1 -5492.373,E2 -5492.373} C_VEL
LIN {X 0,Y 509.277,Z 706.76,A -85,B 0,C 180,E1 -5493.164,E2 -5493.164} C_VEL
LIN {X 0,Y 509.312,Z 703.695,A -85,B 0,C 180,E1 -5494.353,E2 -5494.353} C_VEL
LIN {X 0,Y 509.35,Z 699.596,A -85,B 0,C 180,E1 -5495.543,E2 -5495.543} C_VEL
LIN {X 0,Y 509.421,Z 693.72,A -85,B 0,C 180,E1 -5496.866,E2 -5496.866} C_VEL
LIN {X 0,Y 509.563,Z 686.518,A -85,B 0,C 180,E1 -5498.127,E2 -5498.127} C_VEL
LIN {X 0,Y 509.734,Z 678.012,A -85,B 0,C 180,E1 -5499.323,E2 -5499.323} C_VEL
LIN {X 0,Y 509.992,Z 668.162,A -85,B 0,C 180,E1 -5500.42,E2 -5500.42} C_VEL
LIN {X 0,Y 510.252,Z 658.218,A -85,B 0,C 180,E1 -5501.319,E2 -5501.319} C_VEL
LIN {X 0,Y 510.503,Z 648.25,A -85,B 0,C 180,E1 -5502.051,E2 -5502.051} C_VEL
LIN {X 0,Y 510.769,Z 636.808,A -85,B 0,C 180,E1 -5502.718,E2 -5502.718} C_VEL
LIN {X 0,Y 511.093,Z 623.71,A -85,B 0,C 180,E1 -5503.316,E2 -5503.316} C_VEL
LIN {X 0,Y 511.388,Z 610.582,A -85,B 0,C 180,E1 -5503.739,E2 -5503.739} C_VEL
LIN {X 0,Y 511.611,Z 596.779,A -85,B 0,C 180,E1 -5504.011,E2 -5504.011} C_VEL
LIN {X 0,Y 511.92,Z 507.106,A -85,B 0,C 180,E1 -5505.325,E2 -5505.325} C_VEL
LIN {X 0,Y 510.439,Z 492.668,A -85,B 0,C 180,E1 -5505.608,E2 -5505.608} C_VEL
LIN {X 0,Y 510.856,Z 466.438,A -85,B 0,C 180,E1 -5508.654,E2 -5508.654} C_VEL
LIN {X 0,Y 511.392,Z 440.065,A -85,B 0,C 180,E1 -5511.781,E2 -5511.781} C_VEL
LIN {X 0,Y 512.022,Z 413.999,A -85,B 0,C 180,E1 -5514.943,E2 -5514.943} C_VEL
LIN {X 0,Y 512.413,Z 398.033,A -85,B 0,C 180,E1 -5516.936,E2 -5516.936} C_VEL
LIN {X 0,Y 510.222,Z 386.95,A -85,B 0,C 180,E1 -5518.468,E2 -5518.468} C_VEL
LIN {X 0,Y 509.815,Z 385.085,A -85,B 0,C 180,E1 -5518.781,E2 -5518.781} C_VEL
LIN {X 0,Y 509.788,Z 384.987,A -85,B 0,C 180,E1 -5521.592,E2 -5521.592} C_VEL
LIN {X 0,Y 509.822,Z 384.981,A -85,B 0,C 180,E1 -5524.416,E2 -5524.416} C_VEL
LIN {X 0,Y 509.776,Z 384.985,A -85,B 0,C 180,E1 -5527.344,E2 -5527.344} C_VEL
LIN {X 0,Y 509.786,Z 384.982,A -85,B 0,C 180,E1 -5530.387,E2 -5530.387} C_VEL
LIN {X 0,Y 509.806,Z 384.984,A -85,B 0,C 180,E1 -5533.573,E2 -5533.573} C_VEL
LIN {X 0,Y 509.806,Z 384.978,A -85,B 0,C 180,E1 -5536.427,E2 -5536.427} C_VEL
LIN {X 0,Y 509.814,Z 384.984,A -85,B 0,C 180,E1 -5539.615,E2 -5539.615} C_VEL
LIN {X 0,Y 509.796,Z 384.979,A -85,B 0,C 180,E1 -5542.657,E2 -5542.657} C_VEL
LIN {X 0,Y 509.844,Z 384.979,A -85,B 0,C 180,E1 -5545.8,E2 -5545.8} C_VEL
LIN {X 0,Y 509.848,Z 384.973,A -85,B 0,C 180,E1 -5548.72,E2 -5548.72} C_VEL
LIN {X 0,Y 509.852,Z 384.977,A -85,B 0,C 180,E1 -5551.154,E2 -5551.154} C_VEL
LIN {X 0,Y 509.867,Z 384.973,A -85,B 0,C 180,E1 -5553.827,E2 -5553.827} C_VEL
LIN {X 0,Y 509.824,Z 384.977,A -85,B 0,C 180,E1 -5556.436,E2 -5556.436} C_VEL
LIN {X 0,Y 509.92,Z 384.968,A -85,B 0,C 180,E1 -5559.845,E2 -5559.845} C_VEL
LIN {X 0,Y 509.878,Z 384.976,A -85,B 0,C 180,E1 -5563.174,E2 -5563.174} C_VEL
LIN {X 0,Y 509.933,Z 385.155,A -85,B 0,C 180,E1 -5564.819,E2 -5564.819} C_VEL
LIN {X 0,Y 510.12,Z 385.927,A -85,B 0,C 180,E1 -5564.934,E2 -5564.934} C_VEL
LIN {X 0,Y 512.055,Z 391.731,A -85,B 0,C 180,E1 -5565.113,E2 -5565.113} C_VEL
LIN {X 0,Y 511.654,Z 467.8,A -85,B 0,C 180,E1 -5566.294,E2 -5566.294} C_VEL
LIN {X 0,Y 511.547,Z 481.2,A -85,B 0,C 180,E1 -5566.67,E2 -5566.67} C_VEL
LIN {X 0,Y 511.439,Z 493.823,A -85,B 0,C 180,E1 -5567.198,E2 -5567.198} C_VEL
LIN {X 0,Y 511.234,Z 505.397,A -85,B 0,C 180,E1 -5567.849,E2 -5567.849} C_VEL
LIN {X 0,Y 511.039,Z 515.873,A -85,B 0,C 180,E1 -5568.598,E2 -5568.598} C_VEL
LIN {X 0,Y 510.734,Z 525.999,A -85,B 0,C 180,E1 -5569.495,E2 -5569.495} C_VEL
LIN {X 0,Y 510.529,Z 535.028,A -85,B 0,C 180,E1 -5570.492,E2 -5570.492} C_VEL
LIN {X 0,Y 510.235,Z 543.778,A -85,B 0,C 180,E1 -5571.684,E2 -5571.684} C_VEL
LIN {X 0,Y 509.996,Z 550.777,A -85,B 0,C 180,E1 -5572.876,E2 -5572.876} C_VEL
LIN {X 0,Y 509.93,Z 556.294,A -85,B 0,C 180,E1 -5574.067,E2 -5574.067} C_VEL
LIN {X 0,Y 509.73,Z 560.626,A -85,B 0,C 180,E1 -5575.255,E2 -5575.255} C_VEL
LIN {X 0,Y 509.672,Z 562.889,A -85,B 0,C 180,E1 -5576.047,E2 -5576.047} C_VEL
LIN {X 0,Y 509.707,Z 564.714,A -85,B 0,C 180,E1 -5576.838,E2 -5576.838} C_VEL
LIN {X 0,Y 509.589,Z 566.126,A -85,B 0,C 180,E1 -5577.629,E2 -5577.629} C_VEL
LIN {X 0,Y 509.608,Z 567.083,A -85,B 0,C 180,E1 -5578.42,E2 -5578.42} C_VEL
LIN {X 0,Y 509.54,Z 567.861,A -85,B 0,C 180,E1 -5580,E2 -5580} C_VEL
LIN {X 0,Y 509.554,Z 567.635,A -85,B 0,C 180,E1 -5580.79,E2 -5580.79} C_VEL
LIN {X 0,Y 509.506,Z 567.014,A -85,B 0,C 180,E1 -5581.581,E2 -5581.581} C_VEL
LIN {X 0,Y 509.578,Z 565.989,A -85,B 0,C 180,E1 -5582.371,E2 -5582.371} C_VEL
LIN {X 0,Y 509.569,Z 564.585,A -85,B 0,C 180,E1 -5583.163,E2 -5583.163} C_VEL
LIN {X 0,Y 509.694,Z 561.63,A -85,B 0,C 180,E1 -5584.349,E2 -5584.349} C_VEL
LIN {X 0,Y 509.735,Z 557.656,A -85,B 0,C 180,E1 -5585.538,E2 -5585.538} C_VEL
LIN {X 0,Y 509.915,Z 552.292,A -85,B 0,C 180,E1 -5586.773,E2 -5586.773} C_VEL
LIN {X 0,Y 510.077,Z 546.036,A -85,B 0,C 180,E1 -5587.92,E2 -5587.92} C_VEL
LIN {X 0,Y 510.328,Z 537.953,A -85,B 0,C 180,E1 -5589.113,E2 -5589.113} C_VEL
LIN {X 0,Y 510.485,Z 529.689,A -85,B 0,C 180,E1 -5590.11,E2 -5590.11} C_VEL
LIN {X 0,Y 510.744,Z 519.523,A -85,B 0,C 180,E1 -5591.107,E2 -5591.107} C_VEL
LIN {X 0,Y 511.146,Z 507.742,A -85,B 0,C 180,E1 -5592.019,E2 -5592.019} C_VEL
LIN {X 0,Y 511.274,Z 496.607,A -85,B 0,C 180,E1 -5592.705,E2 -5592.705} C_VEL
LIN {X 0,Y 511.475,Z 484.875,A -85,B 0,C 180,E1 -5593.256,E2 -5593.256} C_VEL
LIN {X 0,Y 511.667,Z 471.378,A -85,B 0,C 180,E1 -5593.706,E2 -5593.706} C_VEL
LIN {X 0,Y 511.711,Z 457.967,A -85,B 0,C 180,E1 -5593.983,E2 -5593.983} C_VEL
LIN {X 0,Y 511.964,Z 391.455,A -85,B 0,C 180,E1 -5594.979,E2 -5594.979} C_VEL
LIN {X 0,Y 510.105,Z 385.943,A -85,B 0,C 180,E1 -5595.137,E2 -5595.137} C_VEL
LIN {X 0,Y 509.907,Z 385.061,A -85,B 0,C 180,E1 -5595.29,E2 -5595.29} C_VEL
LIN {X 0,Y 509.865,Z 384.976,A -85,B 0,C 180,E1 -5598.484,E2 -5598.484} C_VEL
LIN {X 0,Y 509.854,Z 384.978,A -85,B 0,C 180,E1 -5601.002,E2 -5601.002} C_VEL
LIN {X 0,Y 509.865,Z 384.974,A -85,B 0,C 180,E1 -5604.426,E2 -5604.426} C_VEL
LIN {X 0,Y 509.862,Z 384.972,A -85,B 0,C 180,E1 -5607.057,E2 -5607.057} C_VEL
LIN {X 0,Y 509.86,Z 384.967,A -85,B 0,C 180,E1 -5609.751,E2 -5609.751} C_VEL
LIN {X 0,Y 509.87,Z 384.972,A -85,B 0,C 180,E1 -5612.773,E2 -5612.773} C_VEL
LIN {X 0,Y 509.826,Z 384.975,A -85,B 0,C 180,E1 -5615.578,E2 -5615.578} C_VEL
LIN {X 0,Y 509.852,Z 384.973,A -85,B 0,C 180,E1 -5618.338,E2 -5618.338} C_VEL
LIN {X 0,Y 509.855,Z 384.97,A -85,B 0,C 180,E1 -5621.426,E2 -5621.426} C_VEL
LIN {X 0,Y 509.802,Z 384.981,A -85,B 0,C 180,E1 -5622.859,E2 -5622.859} C_VEL
LIN {X 0,Y 509.135,Z 385.066,A -85,B 0,C 180,E1 -5623.518,E2 -5623.518} C_VEL
LIN {X 0,Y 506.274,Z 385.423,A -85,B 0,C 180,E1 -5624.588,E2 -5624.588} C_VEL
LIN {X 0,Y 503.86,Z 385.719,A -85,B 0,C 180,E1 -5625.45,E2 -5625.45} C_VEL
LIN {X 0,Y 502.832,Z 385.847,A -85,B 0,C 180,E1 -5626.116,E2 -5626.116} C_VEL
LIN {X 0,Y 502.753,Z 385.859,A -85,B 0,C 180,E1 -5626.341,E2 -5626.341} C_VEL
LIN {X 0,Y 502.801,Z 385.854,A -85,B 0,C 180,E1 -5629.008,E2 -5629.008} C_VEL
LIN {X 0,Y 502.792,Z 385.846,A -85,B 0,C 180,E1 -5632.046,E2 -5632.046} C_VEL
LIN {X 0,Y 502.8,Z 385.849,A -85,B 0,C 180,E1 -5635.034,E2 -5635.034} C_VEL
LIN {X 0,Y 502.786,Z 385.851,A -85,B 0,C 180,E1 -5637.915,E2 -5637.915} C_VEL
LIN {X 0,Y 502.845,Z 385.867,A -85,B 0,C 180,E1 -5641.172,E2 -5641.172} C_VEL
LIN {X 0,Y 502.901,Z 386.154,A -85,B 0,C 180,E1 -5641.347,E2 -5641.347} C_VEL
LIN {X 0,Y 505.969,Z 399.824,A -85,B 0,C 180,E1 -5643.232,E2 -5643.232} C_VEL
LIN {X 0,Y 505.553,Z 419.968,A -85,B 0,C 180,E1 -5645.789,E2 -5645.789} C_VEL
LIN {X 0,Y 504.788,Z 445.337,A -85,B 0,C 180,E1 -5649,E2 -5649} C_VEL
LIN {X 0,Y 504.157,Z 469.227,A -85,B 0,C 180,E1 -5651.962,E2 -5651.962} C_VEL
LIN {X 0,Y 503.829,Z 488.041,A -85,B 0,C 180,E1 -5654.221,E2 -5654.221} C_VEL
LIN {X 0,Y 505.392,Z 499.515,A -85,B 0,C 180,E1 -5654.453,E2 -5654.453} C_VEL
LIN {X 0,Y 504.869,Z 597.859,A -85,B 0,C 180,E1 -5655.875,E2 -5655.875} C_VEL
LIN {X 0,Y 504.663,Z 611.446,A -85,B 0,C 180,E1 -5656.229,E2 -5656.229} C_VEL
LIN {X 0,Y 504.328,Z 623.563,A -85,B 0,C 180,E1 -5656.707,E2 -5656.707} C_VEL
LIN {X 0,Y 504.018,Z 635.854,A -85,B 0,C 180,E1 -5657.367,E2 -5657.367} C_VEL
LIN {X 0,Y 503.718,Z 646.827,A -85,B 0,C 180,E1 -5658.124,E2 -5658.124} C_VEL
LIN {X 0,Y 503.3,Z 657.3,A -85,B 0,C 180,E1 -5659.032,E2 -5659.032} C_VEL
LIN {X 0,Y 502.973,Z 667.617,A -85,B 0,C 180,E1 -5660.144,E2 -5660.144} C_VEL
LIN {X 0,Y 502.654,Z 676.58,A -85,B 0,C 180,E1 -5661.356,E2 -5661.356} C_VEL
LIN {X 0,Y 502.423,Z 683.777,A -85,B 0,C 180,E1 -5662.566,E2 -5662.566} C_VEL
LIN {X 0,Y 502.313,Z 690.388,A -85,B 0,C 180,E1 -5663.977,E2 -5663.977} C_VEL
LIN {X 0,Y 502.112,Z 694.734,A -85,B 0,C 180,E1 -5665.183,E2 -5665.183} C_VEL
LIN {X 0,Y 502.185,Z 697.02,A -85,B 0,C 180,E1 -5665.988,E2 -5665.988} C_VEL
LIN {X 0,Y 502.123,Z 698.886,A -85,B 0,C 180,E1 -5666.791,E2 -5666.791} C_VEL
LIN {X 0,Y 502.092,Z 700.316,A -85,B 0,C 180,E1 -5667.593,E2 -5667.593} C_VEL
LIN {X 0,Y 501.991,Z 701.936,A -85,B 0,C 180,E1 -5669.198,E2 -5669.198} C_VEL
LIN {X 0,Y 501.98,Z 702.175,A -85,B 0,C 180,E1 -5670,E2 -5670} C_VEL
LIN {X 0,Y 501.99,Z 701.989,A -85,B 0,C 180,E1 -5670.802,E2 -5670.802} C_VEL
LIN {X 0,Y 502.092,Z 700.438,A -85,B 0,C 180,E1 -5672.407,E2 -5672.407} C_VEL
LIN {X 0,Y 502.124,Z 699.076,A -85,B 0,C 180,E1 -5673.21,E2 -5673.21} C_VEL
LIN {X 0,Y 502.156,Z 696.207,A -85,B 0,C 180,E1 -5674.415,E2 -5674.415} C_VEL
LIN {X 0,Y 502.274,Z 692.309,A -85,B 0,C 180,E1 -5675.621,E2 -5675.621} C_VEL
LIN {X 0,Y 502.308,Z 687.264,A -85,B 0,C 180,E1 -5676.83,E2 -5676.83} C_VEL
LIN {X 0,Y 502.515,Z 680.898,A -85,B 0,C 180,E1 -5678.04,E2 -5678.04} C_VEL
LIN {X 0,Y 502.746,Z 672.997,A -85,B 0,C 180,E1 -5679.251,E2 -5679.251} C_VEL
LIN {X 0,Y 503.024,Z 664.932,A -85,B 0,C 180,E1 -5680.261,E2 -5680.261} C_VEL
LIN {X 0,Y 503.424,Z 655.043,A -85,B 0,C 180,E1 -5681.271,E2 -5681.271} C_VEL
LIN {X 0,Y 503.776,Z 644.072,A -85,B 0,C 180,E1 -5682.171,E2 -5682.171} C_VEL
LIN {X 0,Y 504.107,Z 633.101,A -85,B 0,C 180,E1 -5682.889,E2 -5682.889} C_VEL
LIN {X 0,Y 504.45,Z 621.02,A -85,B 0,C 180,E1 -5683.495,E2 -5683.495} C_VEL
LIN {X 0,Y 504.721,Z 607.742,A -85,B 0,C 180,E1 -5683.975,E2 -5683.975} C_VEL
LIN {X 0,Y 504.956,Z 594.428,A -85,B 0,C 180,E1 -5684.277,E2 -5684.277} C_VEL
LIN {X 0,Y 505.361,Z 498.652,A -85,B 0,C 180,E1 -5685.651,E2 -5685.651} C_VEL
LIN {X 0,Y 503.838,Z 488.077,A -85,B 0,C 180,E1 -5685.869,E2 -5685.869} C_VEL
LIN {X 0,Y 504.275,Z 464.67,A -85,B 0,C 180,E1 -5688.696,E2 -5688.696} C_VEL
LIN {X 0,Y 504.968,Z 439.278,A -85,B 0,C 180,E1 -5691.858,E2 -5691.858} C_VEL
LIN {X 0,Y 505.591,Z 417.305,A -85,B 0,C 180,E1 -5694.647,E2 -5694.647} C_VEL
LIN {X 0,Y 506.027,Z 400.46,A -85,B 0,C 180,E1 -5696.781,E2 -5696.781} C_VEL
LIN {X 0,Y 502.837,Z 386.009,A -85,B 0,C 180,E1 -5698.782,E2 -5698.782} C_VEL
LIN {X 0,Y 502.795,Z 385.854,A -85,B 0,C 180,E1 -5701.498,E2 -5701.498} C_VEL
LIN {X 0,Y 502.796,Z 385.854,A -85,B 0,C 180,E1 -5703.995,E2 -5703.995} C_VEL
LIN {X 0,Y 502.74,Z 385.856,A -85,B 0,C 180,E1 -5707.172,E2 -5707.172} C_VEL
LIN {X 0,Y 502.774,Z 385.851,A -85,B 0,C 180,E1 -5710.017,E2 -5710.017} C_VEL
LIN {X 0,Y 502.749,Z 385.86,A -85,B 0,C 180,E1 -5713.234,E2 -5713.234} C_VEL
LIN {X 0,Y 502.782,Z 385.851,A -85,B 0,C 180,E1 -5715.66,E2 -5715.66} C_VEL
LIN {X 0,Y 502.772,Z 385.854,A -85,B 0,C 180,E1 -5719.012,E2 -5719.012} C_VEL
LIN {X 0,Y 502.767,Z 385.854,A -85,B 0,C 180,E1 -5722.044,E2 -5722.044} C_VEL
LIN {X 0,Y 502.791,Z 385.852,A -85,B 0,C 180,E1 -5725.033,E2 -5725.033} C_VEL
LIN {X 0,Y 502.786,Z 385.858,A -85,B 0,C 180,E1 -5727.915,E2 -5727.915} C_VEL
LIN {X 0,Y 502.806,Z 385.846,A -85,B 0,C 180,E1 -5730.711,E2 -5730.711} C_VEL
LIN {X 0,Y 502.777,Z 385.857,A -85,B 0,C 180,E1 -5733.46,E2 -5733.46} C_VEL
LIN {X 0,Y 502.771,Z 385.851,A -85,B 0,C 180,E1 -5736.085,E2 -5736.085} C_VEL
LIN {X 0,Y 502.783,Z 385.852,A -85,B 0,C 180,E1 -5738.689,E2 -5738.689} C_VEL
LIN {X 0,Y 502.811,Z 385.849,A -85,B 0,C 180,E1 -5741.247,E2 -5741.247} C_VEL
LIN {X 0,Y 502.84,Z 385.844,A -85,B 0,C 180,E1 -5744.665,E2 -5744.665} C_VEL
LIN {X 0,Y 502.874,Z 385.836,A -85,B 0,C 180,E1 -5748.043,E2 -5748.043} C_VEL
LIN {X 0,Y 502.845,Z 385.844,A -85,B 0,C 180,E1 -5751.156,E2 -5751.156} C_VEL
LIN {X 0,Y 502.874,Z 385.846,A -85,B 0,C 180,E1 -5753.581,E2 -5753.581} C_VEL
LIN {X 0,Y 502.833,Z 385.841,A -85,B 0,C 180,E1 -5756.795,E2 -5756.795} C_VEL
LIN {X 0,Y 502.895,Z 385.839,A -85,B 0,C 180,E1 -5758.398,E2 -5758.398} C_VEL
LIN {X 0,Y 503.006,Z 385.826,A -85,B 0,C 180,E1 -5760,E2 -5760} C_VEL
LIN {X 0,Y 503.012,Z 385.815,A -85,B 0,C 180,E1 -5762.402,E2 -5762.402} C_VEL
LIN {X 0,Y 502.895,Z 385.843,A -85,B 0,C 180,E1 -5765.614,E2 -5765.614} C_VEL
LIN {X 0,Y 502.85,Z 385.843,A -85,B 0,C 180,E1 -5768.034,E2 -5768.034} C_VEL
LIN {X 0,Y 502.841,Z 385.842,A -85,B 0,C 180,E1 -5771.284,E2 -5771.284} C_VEL
LIN {X 0,Y 502.803,Z 385.847,A -85,B 0,C 180,E1 -5774.572,E2 -5774.572} C_VEL
LIN {X 0,Y 502.791,Z 385.854,A -85,B 0,C 180,E1 -5778.101,E2 -5778.101} C_VEL
LIN {X 0,Y 502.764,Z 385.856,A -85,B 0,C 180,E1 -5781.312,E2 -5781.312} C_VEL
LIN {X 0,Y 502.761,Z 385.856,A -85,B 0,C 180,E1 -5783.915,E2 -5783.915} C_VEL
LIN {X 0,Y 502.76,Z 385.855,A -85,B 0,C 180,E1 -5786.572,E2 -5786.572} C_VEL
LIN {X 0,Y 502.805,Z 385.844,A -85,B 0,C 180,E1 -5789.289,E2 -5789.289} C_VEL
LIN {X 0,Y 502.766,Z 385.858,A -85,B 0,C 180,E1 -5792.086,E2 -5792.086} C_VEL
LIN {X 0,Y 502.785,Z 385.847,A -85,B 0,C 180,E1 -5794.967,E2 -5794.967} C_VEL
LIN {X 0,Y 502.756,Z 385.853,A -85,B 0,C 180,E1 -5798.48,E2 -5798.48} C_VEL
LIN {X 0,Y 502.751,Z 385.84,A -85,B 0,C 180,E1 -5801.073,E2 -5801.073} C_VEL
LIN {X 0,Y 502.78,Z 385.853,A -85,B 0,C 180,E1 -5804.529,E2 -5804.529} C_VEL
LIN {X 0,Y 502.737,Z 385.852,A -85,B 0,C 180,E1 -5807.854,E2 -5807.854} C_VEL
LIN {X 0,Y 502.77,Z 385.852,A -85,B 0,C 180,E1 -5811.021,E2 -5811.021} C_VEL
LIN {X 0,Y 502.744,Z 385.863,A -85,B 0,C 180,E1 -5814.174,E2 -5814.174} C_VEL
LIN {X 0,Y 502.771,Z 385.856,A -85,B 0,C 180,E1 -5817.005,E2 -5817.005} C_VEL
LIN {X 0,Y 502.747,Z 385.864,A -85,B 0,C 180,E1 -5820.079,E2 -5820.079} C_VEL
LIN {X 0,Y 502.809,Z 386.165,A -85,B 0,C 180,E1 -5820.611,E2 -5820.611} C_VEL
LIN {X 0,Y 505.831,Z 399.29,A -85,B 0,C 180,E1 -5822.486,E2 -5822.486} C_VEL
LIN {X 0,Y 506.141,Z 403.272,A -85,B 0,C 180,E1 -5823.015,E2 -5823.015} C_VEL
LIN {X 0,Y 505.303,Z 426.897,A -85,B 0,C 180,E1 -5825.994,E2 -5825.994} C_VEL
LIN {X 0,Y 504.527,Z 451.571,A -85,B 0,C 180,E1 -5829.064,E2 -5829.064} C_VEL
LIN {X 0,Y 503.88,Z 476.8,A -85,B 0,C 180,E1 -5832.13,E2 -5832.13} C_VEL
LIN {X 0,Y 503.523,Z 493.632,A -85,B 0,C 180,E1 -5834.161,E2 -5834.161} C_VEL
LIN {X 0,Y 505.243,Z 510.392,A -85,B 0,C 180,E1 -5834.499,E2 -5834.499} C_VEL
LIN {X 0,Y 504.642,Z 604.516,A -85,B 0,C 180,E1 -5835.919,E2 -5835.919} C_VEL
LIN {X 0,Y 504.321,Z 617.536,A -85,B 0,C 180,E1 -5836.27,E2 -5836.27} C_VEL
LIN {X 0,Y 504.018,Z 629.645,A -85,B 0,C 180,E1 -5836.75,E2 -5836.75} C_VEL
LIN {X 0,Y 503.678,Z 643.999,A -85,B 0,C 180,E1 -5837.512,E2 -5837.512} C_VEL
LIN {X 0,Y 503.42,Z 654.381,A -85,B 0,C 180,E1 -5838.219,E2 -5838.219} C_VEL
LIN {X 0,Y 503.097,Z 665.059,A -85,B 0,C 180,E1 -5839.129,E2 -5839.129} C_VEL
LIN {X 0,Y 502.814,Z 674.65,A -85,B 0,C 180,E1 -5840.141,E2 -5840.141} C_VEL
LIN {X 0,Y 502.585,Z 682.474,A -85,B 0,C 180,E1 -5841.151,E2 -5841.151} C_VEL
LIN {X 0,Y 502.401,Z 690.087,A -85,B 0,C 180,E1 -5842.363,E2 -5842.363} C_VEL
LIN {X 0,Y 502.255,Z 696.188,A -85,B 0,C 180,E1 -5843.573,E2 -5843.573} C_VEL
LIN {X 0,Y 502.225,Z 701,A -85,B 0,C 180,E1 -5844.781,E2 -5844.781} C_VEL
LIN {X 0,Y 502.244,Z 704.673,A -85,B 0,C 180,E1 -5845.988,E2 -5845.988} C_VEL
LIN {X 0,Y 502.186,Z 706.559,A -85,B 0,C 180,E1 -5846.791,E2 -5846.791} C_VEL
LIN {X 0,Y 502.164,Z 707.994,A -85,B 0,C 180,E1 -5847.594,E2 -5847.594} C_VEL
LIN {X 0,Y 502.078,Z 709.61,A -85,B 0,C 180,E1 -5849.198,E2 -5849.198} C_VEL
LIN {X 0,Y 502.095,Z 709.829,A -85,B 0,C 180,E1 -5850,E2 -5850} C_VEL
LIN {X 0,Y 502.104,Z 709.611,A -85,B 0,C 180,E1 -5850.802,E2 -5850.802} C_VEL
LIN {X 0,Y 502.174,Z 707.989,A -85,B 0,C 180,E1 -5852.406,E2 -5852.406} C_VEL
LIN {X 0,Y 502.195,Z 706.567,A -85,B 0,C 180,E1 -5853.209,E2 -5853.209} C_VEL
LIN {X 0,Y 502.208,Z 703.59,A -85,B 0,C 180,E1 -5854.414,E2 -5854.414} C_VEL
LIN {X 0,Y 502.267,Z 699.551,A -85,B 0,C 180,E1 -5855.621,E2 -5855.621} C_VEL
LIN {X 0,Y 502.337,Z 693.416,A -85,B 0,C 180,E1 -5857.011,E2 -5857.011} C_VEL
LIN {X 0,Y 502.52,Z 686.492,A -85,B 0,C 180,E1 -5858.242,E2 -5858.242} C_VEL
LIN {X 0,Y 502.648,Z 679.516,A -85,B 0,C 180,E1 -5859.253,E2 -5859.253} C_VEL
LIN {X 0,Y 502.916,Z 671.068,A -85,B 0,C 180,E1 -5860.263,E2 -5860.263} C_VEL
LIN {X 0,Y 503.184,Z 660.592,A -85,B 0,C 180,E1 -5861.276,E2 -5861.276} C_VEL
LIN {X 0,Y 503.526,Z 650.187,A -85,B 0,C 180,E1 -5862.085,E2 -5862.085} C_VEL
LIN {X 0,Y 503.797,Z 638.751,A -85,B 0,C 180,E1 -5862.79,E2 -5862.79} C_VEL
LIN {X 0,Y 504.084,Z 626.648,A -85,B 0,C 180,E1 -5863.351,E2 -5863.351} C_VEL
LIN {X 0,Y 504.416,Z 610.44,A -85,B 0,C 180,E1 -5863.881,E2 -5863.881} C_VEL
LIN {X 0,Y 504.648,Z 597.389,A -85,B 0,C 180,E1 -5864.157,E2 -5864.157} C_VEL
LIN {X 0,Y 504.988,Z 507.364,A -85,B 0,C 180,E1 -5865.514,E2 -5865.514} C_VEL
LIN {X 0,Y 503.373,Z 491.558,A -85,B 0,C 180,E1 -5865.823,E2 -5865.823} C_VEL
LIN {X 0,Y 503.786,Z 468.588,A -85,B 0,C 180,E1 -5868.524,E2 -5868.524} C_VEL
LIN {X 0,Y 504.373,Z 442.483,A -85,B 0,C 180,E1 -5871.67,E2 -5871.67} C_VEL
LIN {X 0,Y 505.088,Z 415.604,A -85,B 0,C 180,E1 -5874.991,E2 -5874.991} C_VEL
LIN {X 0,Y 505.461,Z 398.729,A -85,B 0,C 180,E1 -5877.143,E2 -5877.143} C_VEL
LIN {X 0,Y 502.789,Z 385.982,A -85,B 0,C 180,E1 -5879.003,E2 -5879.003} C_VEL
LIN {X 0,Y 502.756,Z 385.863,A -85,B 0,C 180,E1 -5882.087,E2 -5882.087} C_VEL
LIN {X 0,Y 502.754,Z 385.859,A -85,B 0,C 180,E1 -5884.97,E2 -5884.97} C_VEL
LIN {X 0,Y 502.755,Z 385.859,A -85,B 0,C 180,E1 -5888.48,E2 -5888.48} C_VEL
LIN {X 0,Y 502.75,Z 385.858,A -85,B 0,C 180,E1 -5891.073,E2 -5891.073} C_VEL
LIN {X 0,Y 502.787,Z 385.853,A -85,B 0,C 180,E1 -5894.53,E2 -5894.53} C_VEL
LIN {X 0,Y 502.767,Z 385.86,A -85,B 0,C 180,E1 -5897.857,E2 -5897.857} C_VEL
LIN {X 0,Y 502.785,Z 385.854,A -85,B 0,C 180,E1 -5901.022,E2 -5901.022} C_VEL
LIN {X 0,Y 502.77,Z 385.857,A -85,B 0,C 180,E1 -5904.17,E2 -5904.17} C_VEL
LIN {X 0,Y 502.833,Z 385.849,A -85,B 0,C 180,E1 -5906.994,E2 -5906.994} C_VEL
LIN {X 0,Y 502.817,Z 385.851,A -85,B 0,C 180,E1 -5910.065,E2 -5910.065} C_VEL
LIN {X 0,Y 502.825,Z 385.854,A -85,B 0,C 180,E1 -5913.449,E2 -5913.449} C_VEL
LIN {X 0,Y 502.775,Z 385.856,A -85,B 0,C 180,E1 -5916.085,E2 -5916.085} C_VEL
LIN {X 0,Y 502.786,Z 385.855,A -85,B 0,C 180,E1 -5918.689,E2 -5918.689} C_VEL
LIN {X 0,Y 502.83,Z 385.854,A -85,B 0,C 180,E1 -5921.248,E2 -5921.248} C_VEL
LIN {X 0,Y 502.86,Z 385.974,A -85,B 0,C 180,E1 -5924.575,E2 -5924.575} C_VEL
LIN {X 0,Y 503.052,Z 386.857,A -85,B 0,C 180,E1 -5924.716,E2 -5924.716} C_VEL
LIN {X 0,Y 505.206,Z 393.009,A -85,B 0,C 180,E1 -5924.91,E2 -5924.91} C_VEL
LIN {X 0,Y 504.756,Z 469.064,A -85,B 0,C 180,E1 -5926.128,E2 -5926.128} C_VEL
LIN {X 0,Y 504.662,Z 482.406,A -85,B 0,C 180,E1 -5926.511,E2 -5926.511} C_VEL
LIN {X 0,Y 504.575,Z 494.51,A -85,B 0,C 180,E1 -5927.021,E2 -5927.021} C_VEL
LIN {X 0,Y 504.358,Z 506.375,A -85,B 0,C 180,E1 -5927.693,E2 -5927.693} C_VEL
LIN {X 0,Y 504.111,Z 517.996,A -85,B 0,C 180,E1 -5928.541,E2 -5928.541} C_VEL
LIN {X 0,Y 503.813,Z 526.906,A -85,B 0,C 180,E1 -5929.349,E2 -5929.349} C_VEL
LIN {X 0,Y 503.592,Z 535.981,A -85,B 0,C 180,E1 -5930.359,E2 -5930.359} C_VEL
LIN {X 0,Y 503.301,Z 544.758,A -85,B 0,C 180,E1 -5931.569,E2 -5931.569} C_VEL
LIN {X 0,Y 503.023,Z 551.782,A -85,B 0,C 180,E1 -5932.776,E2 -5932.776} C_VEL
LIN {X 0,Y 502.95,Z 557.309,A -85,B 0,C 180,E1 -5933.984,E2 -5933.984} C_VEL
LIN {X 0,Y 502.729,Z 561.647,A -85,B 0,C 180,E1 -5935.189,E2 -5935.189} C_VEL
LIN {X 0,Y 502.663,Z 563.91,A -85,B 0,C 180,E1 -5935.991,E2 -5935.991} C_VEL
LIN {X 0,Y 502.707,Z 565.732,A -85,B 0,C 180,E1 -5936.794,E2 -5936.794} C_VEL
LIN {X 0,Y 502.581,Z 567.145,A -85,B 0,C 180,E1 -5937.596,E2 -5937.596} C_VEL
LIN {X 0,Y 502.6,Z 568.096,A -85,B 0,C 180,E1 -5938.397,E2 -5938.397} C_VEL
LIN {X 0,Y 502.523,Z 568.863,A -85,B 0,C 180,E1 -5940,E2 -5940} C_VEL
LIN {X 0,Y 502.538,Z 568.628,A -85,B 0,C 180,E1 -5940.801,E2 -5940.801} C_VEL
LIN {X 0,Y 502.483,Z 567.994,A -85,B 0,C 180,E1 -5941.603,E2 -5941.603} C_VEL
LIN {X 0,Y 502.565,Z 566.958,A -85,B 0,C 180,E1 -5942.404,E2 -5942.404} C_VEL
LIN {X 0,Y 502.544,Z 565.543,A -85,B 0,C 180,E1 -5943.207,E2 -5943.207} C_VEL
LIN {X 0,Y 502.679,Z 562.563,A -85,B 0,C 180,E1 -5944.41,E2 -5944.41} C_VEL
LIN {X 0,Y 502.738,Z 558.558,A -85,B 0,C 180,E1 -5945.616,E2 -5945.616} C_VEL
LIN {X 0,Y 502.936,Z 553.159,A -85,B 0,C 180,E1 -5946.866,E2 -5946.866} C_VEL
LIN {X 0,Y 503.115,Z 546.854,A -85,B 0,C 180,E1 -5948.03,E2 -5948.03} C_VEL
LIN {X 0,Y 503.382,Z 538.721,A -85,B 0,C 180,E1 -5949.239,E2 -5949.239} C_VEL
LIN {X 0,Y 503.552,Z 530.406,A -85,B 0,C 180,E1 -5950.25,E2 -5950.25} C_VEL
LIN {X 0,Y 503.829,Z 520.151,A -85,B 0,C 180,E1 -5951.262,E2 -5951.262} C_VEL
LIN {X 0,Y 504.23,Z 508.401,A -85,B 0,C 180,E1 -5952.179,E2 -5952.179} C_VEL
LIN {X 0,Y 504.365,Z 497.031,A -85,B 0,C 180,E1 -5952.882,E2 -5952.882} C_VEL
LIN {X 0,Y 504.578,Z 485.105,A -85,B 0,C 180,E1 -5953.44,E2 -5953.44} C_VEL
LIN {X 0,Y 504.758,Z 471.357,A -85,B 0,C 180,E1 -5953.897,E2 -5953.897} C_VEL
LIN {X 0,Y 504.815,Z 458.918,A -85,B 0,C 180,E1 -5954.153,E2 -5954.153} C_VEL
LIN {X 0,Y 505.115,Z 392.888,A -85,B 0,C 180,E1 -5955.161,E2 -5955.161} C_VEL
LIN {X 0,Y 503.02,Z 386.712,A -85,B 0,C 180,E1 -5955.346,E2 -5955.346} C_VEL
LIN {X 0,Y 502.84,Z 385.922,A -85,B 0,C 180,E1 -5955.504,E2 -5955.504} C_VEL
LIN {X 0,Y 502.83,Z 385.854,A -85,B 0,C 180,E1 -5958.752,E2 -5958.752} C_VEL
LIN {X 0,Y 502.787,Z 385.855,A -85,B 0,C 180,E1 -5961.311,E2 -5961.311} C_VEL
LIN {X 0,Y 502.787,Z 385.852,A -85,B 0,C 180,E1 -5963.914,E2 -5963.914} C_VEL
LIN {X 0,Y 502.838,Z 385.851,A -85,B 0,C 180,E1 -5966.568,E2 -5966.568} C_VEL
LIN {X 0,Y 502.818,Z 385.845,A -85,B 0,C 180,E1 -5969.935,E2 -5969.935} C_VEL
LIN {X 0,Y 502.832,Z 385.845,A -85,B 0,C 180,E1 -5973.031,E2 -5973.031} C_VEL
LIN {X 0,Y 502.774,Z 385.854,A -85,B 0,C 180,E1 -5975.951,E2 -5975.951} C_VEL
LIN {X 0,Y 502.803,Z 385.854,A -85,B 0,C 180,E1 -5978.976,E2 -5978.976} C_VEL
LIN {X 0,Y 502.806,Z 385.85,A -85,B 0,C 180,E1 -5982.199,E2 -5982.199} C_VEL
LIN {X 0,Y 502.788,Z 385.85,A -85,B 0,C 180,E1 -5985.47,E2 -5985.47} C_VEL
LIN {X 0,Y 502.753,Z 385.859,A -85,B 0,C 180,E1 -5986.341,E2 -5986.341} C_VEL
LIN {X 0,Y 502.097,Z 385.947,A -85,B 0,C 180,E1 -5987.011,E2 -5987.011} C_VEL
LIN {X 0,Y 499.245,Z 386.3,A -85,B 0,C 180,E1 -5988.097,E2 -5988.097} C_VEL
LIN {X 0,Y 496.841,Z 386.597,A -85,B 0,C 180,E1 -5988.973,E2 -5988.973} C_VEL
LIN {X 0,Y 495.827,Z 386.72,A -85,B 0,C 180,E1 -5989.649,E2 -5989.649} C_VEL
LIN {X 0,Y 495.755,Z 386.729,A -85,B 0,C 180,E1 -5989.878,E2 -5989.878} C_VEL
LIN {X 0,Y 495.721,Z 386.733,A -85,B 0,C 180,E1 -5992.555,E2 -5992.555} C_VEL
LIN {X 0,Y 495.779,Z 386.724,A -85,B 0,C 180,E1 -5995.457,E2 -5995.457} C_VEL
LIN {X 0,Y 495.757,Z 386.73,A -85,B 0,C 180,E1 -5998.364,E2 -5998.364} C_VEL
LIN {X 0,Y 495.84,Z 386.94,A -85,B 0,C 180,E1 -6001.088,E2 -6001.088} C_VEL
LIN {X 0,Y 498.982,Z 400.883,A -85,B 0,C 180,E1 -6003.036,E2 -6003.036} C_VEL
LIN {X 0,Y 499.047,Z 407.508,A -85,B 0,C 180,E1 -6003.89,E2 -6003.89} C_VEL
LIN {X 0,Y 498.378,Z 429.716,A -85,B 0,C 180,E1 -6006.743,E2 -6006.743} C_VEL
LIN {X 0,Y 497.752,Z 449.974,A -85,B 0,C 180,E1 -6009.33,E2 -6009.33} C_VEL
LIN {X 0,Y 497.108,Z 475.585,A -85,B 0,C 180,E1 -6012.517,E2 -6012.517} C_VEL
LIN {X 0,Y 496.889,Z 488.224,A -85,B 0,C 180,E1 -6014.006,E2 -6014.006} C_VEL
LIN {X 0,Y 498.552,Z 500.106,A -85,B 0,C 180,E1 -6014.243,E2 -6014.243} C_VEL
LIN {X 0,Y 497.999,Z 597.799,A -85,B 0,C 180,E1 -6015.676,E2 -6015.676} C_VEL
LIN {X 0,Y 497.752,Z 611.438,A -85,B 0,C 180,E1 -6016.034,E2 -6016.034} C_VEL
LIN {X 0,Y 497.439,Z 623.58,A -85,B 0,C 180,E1 -6016.519,E2 -6016.519} C_VEL
LIN {X 0,Y 497.09,Z 636.016,A -85,B 0,C 180,E1 -6017.196,E2 -6017.196} C_VEL
LIN {X 0,Y 496.766,Z 646.865,A -85,B 0,C 180,E1 -6017.955,E2 -6017.955} C_VEL
LIN {X 0,Y 496.321,Z 657.343,A -85,B 0,C 180,E1 -6018.876,E2 -6018.876} C_VEL
LIN {X 0,Y 495.973,Z 667.664,A -85,B 0,C 180,E1 -6020.004,E2 -6020.004} C_VEL
LIN {X 0,Y 495.623,Z 676.63,A -85,B 0,C 180,E1 -6021.232,E2 -6021.232} C_VEL
LIN {X 0,Y 495.349,Z 683.829,A -85,B 0,C 180,E1 -6022.459,E2 -6022.459} C_VEL
LIN {X 0,Y 495.241,Z 690.442,A -85,B 0,C 180,E1 -6023.89,E2 -6023.89} C_VEL
LIN {X 0,Y 495.04,Z 694.788,A -85,B 0,C 180,E1 -6025.114,E2 -6025.114} C_VEL
LIN {X 0,Y 495.083,Z 697.074,A -85,B 0,C 180,E1 -6025.93,E2 -6025.93} C_VEL
LIN {X 0,Y 495.047,Z 698.941,A -85,B 0,C 180,E1 -6026.745,E2 -6026.745} C_VEL
LIN {X 0,Y 494.998,Z 700.371,A -85,B 0,C 180,E1 -6027.559,E2 -6027.559} C_VEL
LIN {X 0,Y 494.911,Z 701.991,A -85,B 0,C 180,E1 -6029.186,E2 -6029.186} C_VEL
LIN {X 0,Y 494.898,Z 702.229,A -85,B 0,C 180,E1 -6030,E2 -6030} C_VEL
LIN {X 0,Y 494.911,Z 702.042,A -85,B 0,C 180,E1 -6030.814,E2 -6030.814} C_VEL
LIN {X 0,Y 494.999,Z 700.491,A -85,B 0,C 180,E1 -6032.441,E2 -6032.441} C_VEL
LIN {X 0,Y 495.047,Z 699.128,A -85,B 0,C 180,E1 -6033.256,E2 -6033.256} C_VEL
LIN {X 0,Y 495.052,Z 696.258,A -85,B 0,C 180,E1 -6034.478,E2 -6034.478} C_VEL
LIN {X 0,Y 495.197,Z 691.253,A -85,B 0,C 180,E1 -6035.99,E2 -6035.99} C_VEL
LIN {X 0,Y 495.277,Z 685.339,A -85,B 0,C 180,E1 -6037.337,E2 -6037.337} C_VEL
LIN {X 0,Y 495.547,Z 678.517,A -85,B 0,C 180,E1 -6038.564,E2 -6038.564} C_VEL
LIN {X 0,Y 495.86,Z 669.983,A -85,B 0,C 180,E1 -6039.793,E2 -6039.793} C_VEL
LIN {X 0,Y 496.206,Z 661.251,A -85,B 0,C 180,E1 -6040.817,E2 -6040.817} C_VEL
LIN {X 0,Y 496.603,Z 651.669,A -85,B 0,C 180,E1 -6041.738,E2 -6041.738} C_VEL
LIN {X 0,Y 496.88,Z 640.688,A -85,B 0,C 180,E1 -6042.589,E2 -6042.589} C_VEL
LIN {X 0,Y 497.285,Z 629.411,A -85,B 0,C 180,E1 -6043.277,E2 -6043.277} C_VEL
LIN {X 0,Y 497.625,Z 617.37,A -85,B 0,C 180,E1 -6043.84,E2 -6043.84} C_VEL
LIN {X 0,Y 497.935,Z 604.939,A -85,B 0,C 180,E1 -6044.248,E2 -6044.248} C_VEL
LIN {X 0,Y 498.129,Z 590.903,A -85,B 0,C 180,E1 -6044.529,E2 -6044.529} C_VEL
LIN {X 0,Y 498.464,Z 499.123,A -85,B 0,C 180,E1 -6045.864,E2 -6045.864} C_VEL
LIN {X 0,Y 496.879,Z 488.084,A -85,B 0,C 180,E1 -6046.092,E2 -6046.092} C_VEL
LIN {X 0,Y 497.3,Z 467.069,A -85,B 0,C 180,E1 -6048.623,E2 -6048.623} C_VEL
LIN {X 0,Y 498.005,Z 442.274,A -85,B 0,C 180,E1 -6051.744,E2 -6051.744} C_VEL
LIN {X 0,Y 498.672,Z 420.259,A -85,B 0,C 180,E1 -6054.567,E2 -6054.567} C_VEL
LIN {X 0,Y 499.14,Z 401.811,A -85,B 0,C 180,E1 -6056.928,E2 -6056.928} C_VEL
LIN {X 0,Y 495.802,Z 386.905,A -85,B 0,C 180,E1 -6059.016,E2 -6059.016} C_VEL
LIN {X 0,Y 495.757,Z 386.73,A -85,B 0,C 180,E1 -6061.725,E2 -6061.725} C_VEL
LIN {X 0,Y 495.763,Z 386.729,A -85,B 0,C 180,E1 -6064.692,E2 -6064.692} C_VEL
LIN {X 0,Y 495.704,Z 386.737,A -85,B 0,C 180,E1 -6067.564,E2 -6067.564} C_VEL
LIN {X 0,Y 495.747,Z 386.725,A -85,B 0,C 180,E1 -6070.045,E2 -6070.045} C_VEL
LIN {X 0,Y 495.698,Z 386.736,A -85,B 0,C 180,E1 -6072.887,E2 -6072.887} C_VEL
LIN {X 0,Y 495.726,Z 386.735,A -85,B 0,C 180,E1 -6075.998,E2 -6075.998} C_VEL
LIN {X 0,Y 495.733,Z 386.734,A -85,B 0,C 180,E1 -6079.297,E2 -6079.297} C_VEL
LIN {X 0,Y 495.728,Z 386.737,A -85,B 0,C 180,E1 -6081.406,E2 -6081.406} C_VEL
LIN {X 0,Y 495.741,Z 386.73,A -85,B 0,C 180,E1 -6084.462,E2 -6084.462} C_VEL
LIN {X 0,Y 495.756,Z 386.727,A -85,B 0,C 180,E1 -6087.405,E2 -6087.405} C_VEL
LIN {X 0,Y 495.76,Z 386.725,A -85,B 0,C 180,E1 -6090.253,E2 -6090.253} C_VEL
LIN {X 0,Y 495.742,Z 386.732,A -85,B 0,C 180,E1 -6093.271,E2 -6093.271} C_VEL
LIN {X 0,Y 495.743,Z 386.723,A -85,B 0,C 180,E1 -6096.612,E2 -6096.612} C_VEL
LIN {X 0,Y 495.783,Z 386.727,A -85,B 0,C 180,E1 -6099.324,E2 -6099.324} C_VEL
LIN {X 0,Y 495.783,Z 386.723,A -85,B 0,C 180,E1 -6101.828,E2 -6101.828} C_VEL
LIN {X 0,Y 495.784,Z 386.725,A -85,B 0,C 180,E1 -6105.217,E2 -6105.217} C_VEL
LIN {X 0,Y 495.825,Z 386.709,A -85,B 0,C 180,E1 -6108.554,E2 -6108.554} C_VEL
LIN {X 0,Y 495.816,Z 386.726,A -85,B 0,C 180,E1 -6111.851,E2 -6111.851} C_VEL
LIN {X 0,Y 495.857,Z 386.709,A -85,B 0,C 180,E1 -6114.306,E2 -6114.306} C_VEL
LIN {X 0,Y 495.978,Z 386.701,A -85,B 0,C 180,E1 -6117.564,E2 -6117.564} C_VEL
LIN {X 0,Y 495.975,Z 386.702,A -85,B 0,C 180,E1 -6120,E2 -6120} C_VEL
LIN {X 0,Y 495.979,Z 386.691,A -85,B 0,C 180,E1 -6122.436,E2 -6122.436} C_VEL
LIN {X 0,Y 495.854,Z 386.721,A -85,B 0,C 180,E1 -6125.694,E2 -6125.694} C_VEL
LIN {X 0,Y 495.814,Z 386.717,A -85,B 0,C 180,E1 -6128.149,E2 -6128.149} C_VEL
LIN {X 0,Y 495.825,Z 386.717,A -85,B 0,C 180,E1 -6131.446,E2 -6131.446} C_VEL
LIN {X 0,Y 495.758,Z 386.724,A -85,B 0,C 180,E1 -6134.784,E2 -6134.784} C_VEL
LIN {X 0,Y 495.751,Z 386.73,A -85,B 0,C 180,E1 -6138.226,E2 -6138.226} C_VEL
LIN {X 0,Y 495.731,Z 386.736,A -85,B 0,C 180,E1 -6141.63,E2 -6141.63} C_VEL
LIN {X 0,Y 495.708,Z 386.734,A -85,B 0,C 180,E1 -6144.277,E2 -6144.277} C_VEL
LIN {X 0,Y 495.721,Z 386.731,A -85,B 0,C 180,E1 -6146.98,E2 -6146.98} C_VEL
LIN {X 0,Y 495.76,Z 386.73,A -85,B 0,C 180,E1 -6150.145,E2 -6150.145} C_VEL
LIN {X 0,Y 495.751,Z 386.728,A -85,B 0,C 180,E1 -6153.236,E2 -6153.236} C_VEL
LIN {X 0,Y 495.689,Z 386.741,A -85,B 0,C 180,E1 -6156.083,E2 -6156.083} C_VEL
LIN {X 0,Y 495.731,Z 386.726,A -85,B 0,C 180,E1 -6158.763,E2 -6158.763} C_VEL
LIN {X 0,Y 495.702,Z 386.719,A -85,B 0,C 180,E1 -6161.787,E2 -6161.787} C_VEL
LIN {X 0,Y 495.733,Z 386.731,A -85,B 0,C 180,E1 -6165.142,E2 -6165.142} C_VEL
LIN {X 0,Y 495.703,Z 386.721,A -85,B 0,C 180,E1 -6168.213,E2 -6168.213} C_VEL
LIN {X 0,Y 495.715,Z 386.733,A -85,B 0,C 180,E1 -6171.405,E2 -6171.405} C_VEL
LIN {X 0,Y 495.716,Z 386.736,A -85,B 0,C 180,E1 -6174.459,E2 -6174.459} C_VEL
LIN {X 0,Y 495.726,Z 386.736,A -85,B 0,C 180,E1 -6177.402,E2 -6177.402} C_VEL
LIN {X 0,Y 495.766,Z 386.967,A -85,B 0,C 180,E1 -6180.356,E2 -6180.356} C_VEL
LIN {X 0,Y 499.141,Z 401.8,A -85,B 0,C 180,E1 -6182.506,E2 -6182.506} C_VEL
LIN {X 0,Y 499.028,Z 410.698,A -85,B 0,C 180,E1 -6183.664,E2 -6183.664} C_VEL
LIN {X 0,Y 498.287,Z 430.846,A -85,B 0,C 180,E1 -6186.234,E2 -6186.234} C_VEL
LIN {X 0,Y 497.485,Z 454.224,A -85,B 0,C 180,E1 -6189.177,E2 -6189.177} C_VEL
LIN {X 0,Y 496.843,Z 477.7,A -85,B 0,C 180,E1 -6192.081,E2 -6192.081} C_VEL
LIN {X 0,Y 496.505,Z 492.86,A -85,B 0,C 180,E1 -6193.934,E2 -6193.934} C_VEL
LIN {X 0,Y 498.376,Z 510.086,A -85,B 0,C 180,E1 -6194.291,E2 -6194.291} C_VEL
LIN {X 0,Y 497.693,Z 603.992,A -85,B 0,C 180,E1 -6195.745,E2 -6195.745} C_VEL
LIN {X 0,Y 497.363,Z 616.898,A -85,B 0,C 180,E1 -6196.1,E2 -6196.1} C_VEL
LIN {X 0,Y 497.053,Z 631.407,A -85,B 0,C 180,E1 -6196.665,E2 -6196.665} C_VEL
LIN {X 0,Y 496.783,Z 642.744,A -85,B 0,C 180,E1 -6197.26,E2 -6197.26} C_VEL
LIN {X 0,Y 496.491,Z 653.002,A -85,B 0,C 180,E1 -6197.948,E2 -6197.948} C_VEL
LIN {X 0,Y 496.093,Z 663.954,A -85,B 0,C 180,E1 -6198.871,E2 -6198.871} C_VEL
LIN {X 0,Y 495.862,Z 672.829,A -85,B 0,C 180,E1 -6199.795,E2 -6199.795} C_VEL
LIN {X 0,Y 495.575,Z 680.952,A -85,B 0,C 180,E1 -6200.82,E2 -6200.82} C_VEL
LIN {X 0,Y 495.376,Z 688.9,A -85,B 0,C 180,E1 -6202.049,E2 -6202.049} C_VEL
LIN {X 0,Y 495.251,Z 694.266,A -85,B 0,C 180,E1 -6203.072,E2 -6203.072} C_VEL
LIN {X 0,Y 495.179,Z 699.496,A -85,B 0,C 180,E1 -6204.298,E2 -6204.298} C_VEL
LIN {X 0,Y 495.081,Z 703.533,A -85,B 0,C 180,E1 -6205.522,E2 -6205.522} C_VEL
LIN {X 0,Y 495.106,Z 706.506,A -85,B 0,C 180,E1 -6206.745,E2 -6206.745} C_VEL
LIN {X 0,Y 495.067,Z 707.934,A -85,B 0,C 180,E1 -6207.559,E2 -6207.559} C_VEL
LIN {X 0,Y 494.993,Z 709.555,A -85,B 0,C 180,E1 -6209.186,E2 -6209.186} C_VEL
LIN {X 0,Y 495.007,Z 709.775,A -85,B 0,C 180,E1 -6210,E2 -6210} C_VEL
LIN {X 0,Y 495.017,Z 709.555,A -85,B 0,C 180,E1 -6210.813,E2 -6210.813} C_VEL
LIN {X 0,Y 495.076,Z 707.935,A -85,B 0,C 180,E1 -6212.441,E2 -6212.441} C_VEL
LIN {X 0,Y 495.115,Z 706.508,A -85,B 0,C 180,E1 -6213.255,E2 -6213.255} C_VEL
LIN {X 0,Y 495.109,Z 703.536,A -85,B 0,C 180,E1 -6214.478,E2 -6214.478} C_VEL
LIN {X 0,Y 495.187,Z 699.497,A -85,B 0,C 180,E1 -6215.702,E2 -6215.702} C_VEL
LIN {X 0,Y 495.252,Z 693.361,A -85,B 0,C 180,E1 -6217.112,E2 -6217.112} C_VEL
LIN {X 0,Y 495.462,Z 686.45,A -85,B 0,C 180,E1 -6218.36,E2 -6218.36} C_VEL
LIN {X 0,Y 495.612,Z 679.471,A -85,B 0,C 180,E1 -6219.385,E2 -6219.385} C_VEL
LIN {X 0,Y 495.893,Z 671.028,A -85,B 0,C 180,E1 -6220.41,E2 -6220.41} C_VEL
LIN {X 0,Y 496.212,Z 660.558,A -85,B 0,C 180,E1 -6221.437,E2 -6221.437} C_VEL
LIN {X 0,Y 496.558,Z 650.16,A -85,B 0,C 180,E1 -6222.257,E2 -6222.257} C_VEL
LIN {X 0,Y 496.864,Z 638.649,A -85,B 0,C 180,E1 -6222.976,E2 -6222.976} C_VEL
LIN {X 0,Y 497.185,Z 626.628,A -85,B 0,C 180,E1 -6223.54,E2 -6223.54} C_VEL
LIN {X 0,Y 497.437,Z 613.515,A -85,B 0,C 180,E1 -6223.976,E2 -6223.976} C_VEL
LIN {X 0,Y 497.696,Z 594.743,A -85,B 0,C 180,E1 -6224.359,E2 -6224.359} C_VEL
LIN {X 0,Y 498.129,Z 508.277,A -85,B 0,C 180,E1 -6225.695,E2 -6225.695} C_VEL
LIN {X 0,Y 496.315,Z 490.22,A -85,B 0,C 180,E1 -6226.064,E2 -6226.064} C_VEL
LIN {X 0,Y 496.781,Z 466.92,A -85,B 0,C 180,E1 -6228.855,E2 -6228.855} C_VEL
LIN {X 0,Y 497.416,Z 441.446,A -85,B 0,C 180,E1 -6231.988,E2 -6231.988} C_VEL
LIN {X 0,Y 498.198,Z 414.835,A -85,B 0,C 180,E1 -6235.349,E2 -6235.349} C_VEL
LIN {X 0,Y 498.664,Z 401.317,A -85,B 0,C 180,E1 -6237.107,E2 -6237.107} C_VEL
LIN {X 0,Y 496.422,Z 389.885,A -85,B 0,C 180,E1 -6238.774,E2 -6238.774} C_VEL
LIN {X 0,Y 495.735,Z 386.831,A -85,B 0,C 180,E1 -6239.282,E2 -6239.282} C_VEL
LIN {X 0,Y 495.725,Z 386.736,A -85,B 0,C 180,E1 -6242.598,E2 -6242.598} C_VEL
LIN {X 0,Y 495.716,Z 386.738,A -85,B 0,C 180,E1 -6245.54,E2 -6245.54} C_VEL
LIN {X 0,Y 495.73,Z 386.733,A -85,B 0,C 180,E1 -6248.763,E2 -6248.763} C_VEL
LIN {X 0,Y 495.702,Z 386.741,A -85,B 0,C 180,E1 -6251.787,E2 -6251.787} C_VEL
LIN {X 0,Y 495.738,Z 386.732,A -85,B 0,C 180,E1 -6255.141,E2 -6255.141} C_VEL
LIN {X 0,Y 495.724,Z 386.734,A -85,B 0,C 180,E1 -6258.215,E2 -6258.215} C_VEL
LIN {X 0,Y 495.742,Z 386.733,A -85,B 0,C 180,E1 -6261.235,E2 -6261.235} C_VEL
LIN {X 0,Y 495.744,Z 386.731,A -85,B 0,C 180,E1 -6264.462,E2 -6264.462} C_VEL
LIN {X 0,Y 495.768,Z 386.732,A -85,B 0,C 180,E1 -6267.406,E2 -6267.406} C_VEL
LIN {X 0,Y 495.765,Z 386.728,A -85,B 0,C 180,E1 -6270.254,E2 -6270.254} C_VEL
LIN {X 0,Y 495.776,Z 386.73,A -85,B 0,C 180,E1 -6273.262,E2 -6273.262} C_VEL
LIN {X 0,Y 495.744,Z 386.732,A -85,B 0,C 180,E1 -6276.613,E2 -6276.613} C_VEL
LIN {X 0,Y 495.781,Z 386.731,A -85,B 0,C 180,E1 -6279.324,E2 -6279.324} C_VEL
LIN {X 0,Y 495.784,Z 386.731,A -85,B 0,C 180,E1 -6281.829,E2 -6281.829} C_VEL
LIN {X 0,Y 495.813,Z 386.829,A -85,B 0,C 180,E1 -6284.323,E2 -6284.323} C_VEL
LIN {X 0,Y 495.996,Z 387.774,A -85,B 0,C 180,E1 -6284.478,E2 -6284.478} C_VEL
LIN {X 0,Y 498.462,Z 394.768,A -85,B 0,C 180,E1 -6284.709,E2 -6284.709} C_VEL
LIN {X 0,Y 497.886,Z 469.654,A -85,B 0,C 180,E1 -6285.933,E2 -6285.933} C_VEL
LIN {X 0,Y 497.795,Z 483.109,A -85,B 0,C 180,E1 -6286.321,E2 -6286.321} C_VEL
LIN {X 0,Y 497.721,Z 495.305,A -85,B 0,C 180,E1 -6286.839,E2 -6286.839} C_VEL
LIN {X 0,Y 497.468,Z 505.677,A -85,B 0,C 180,E1 -6287.418,E2 -6287.418} C_VEL
LIN {X 0,Y 497.233,Z 516.318,A -85,B 0,C 180,E1 -6288.174,E2 -6288.174} C_VEL
LIN {X 0,Y 496.927,Z 526.751,A -85,B 0,C 180,E1 -6289.096,E2 -6289.096} C_VEL
LIN {X 0,Y 496.687,Z 535.254,A -85,B 0,C 180,E1 -6290.018,E2 -6290.018} C_VEL
LIN {X 0,Y 496.398,Z 543.05,A -85,B 0,C 180,E1 -6291.04,E2 -6291.04} C_VEL
LIN {X 0,Y 496.199,Z 550.601,A -85,B 0,C 180,E1 -6292.268,E2 -6292.268} C_VEL
LIN {X 0,Y 496.05,Z 556.599,A -85,B 0,C 180,E1 -6293.492,E2 -6293.492} C_VEL
LIN {X 0,Y 495.838,Z 561.336,A -85,B 0,C 180,E1 -6294.714,E2 -6294.714} C_VEL
LIN {X 0,Y 495.656,Z 564.946,A -85,B 0,C 180,E1 -6295.935,E2 -6295.935} C_VEL
LIN {X 0,Y 495.706,Z 566.764,A -85,B 0,C 180,E1 -6296.749,E2 -6296.749} C_VEL
LIN {X 0,Y 495.571,Z 568.177,A -85,B 0,C 180,E1 -6297.562,E2 -6297.562} C_VEL
LIN {X 0,Y 495.591,Z 569.123,A -85,B 0,C 180,E1 -6298.375,E2 -6298.375} C_VEL
LIN {X 0,Y 495.506,Z 569.874,A -85,B 0,C 180,E1 -6300,E2 -6300} C_VEL
LIN {X 0,Y 495.522,Z 569.626,A -85,B 0,C 180,E1 -6300.813,E2 -6300.813} C_VEL
LIN {X 0,Y 495.461,Z 568.982,A -85,B 0,C 180,E1 -6301.626,E2 -6301.626} C_VEL
LIN {X 0,Y 495.551,Z 567.931,A -85,B 0,C 180,E1 -6302.439,E2 -6302.439} C_VEL
LIN {X 0,Y 495.519,Z 566.495,A -85,B 0,C 180,E1 -6303.252,E2 -6303.252} C_VEL
LIN {X 0,Y 495.663,Z 563.485,A -85,B 0,C 180,E1 -6304.473,E2 -6304.473} C_VEL
LIN {X 0,Y 495.741,Z 559.441,A -85,B 0,C 180,E1 -6305.695,E2 -6305.695} C_VEL
LIN {X 0,Y 495.958,Z 553.998,A -85,B 0,C 180,E1 -6306.962,E2 -6306.962} C_VEL
LIN {X 0,Y 496.172,Z 546.404,A -85,B 0,C 180,E1 -6308.348,E2 -6308.348} C_VEL
LIN {X 0,Y 496.483,Z 537.915,A -85,B 0,C 180,E1 -6309.574,E2 -6309.574} C_VEL
LIN {X 0,Y 496.68,Z 529.163,A -85,B 0,C 180,E1 -6310.6,E2 -6310.6} C_VEL
LIN {X 0,Y 497.014,Z 519.536,A -85,B 0,C 180,E1 -6311.521,E2 -6311.521} C_VEL
LIN {X 0,Y 497.309,Z 508.985,A -85,B 0,C 180,E1 -6312.343,E2 -6312.343} C_VEL
LIN {X 0,Y 497.45,Z 497.337,A -85,B 0,C 180,E1 -6313.065,E2 -6313.065} C_VEL
LIN {X 0,Y 497.669,Z 485.218,A -85,B 0,C 180,E1 -6313.631,E2 -6313.631} C_VEL
LIN {X 0,Y 497.862,Z 472.086,A -85,B 0,C 180,E1 -6314.068,E2 -6314.068} C_VEL
LIN {X 0,Y 497.901,Z 459.55,A -85,B 0,C 180,E1 -6314.327,E2 -6314.327} C_VEL
LIN {X 0,Y 498.283,Z 394.433,A -85,B 0,C 180,E1 -6315.345,E2 -6315.345} C_VEL
LIN {X 0,Y 495.929,Z 387.514,A -85,B 0,C 180,E1 -6315.557,E2 -6315.557} C_VEL
LIN {X 0,Y 495.799,Z 386.78,A -85,B 0,C 180,E1 -6315.73,E2 -6315.73} C_VEL
LIN {X 0,Y 495.785,Z 386.731,A -85,B 0,C 180,E1 -6319.028,E2 -6319.028} C_VEL
LIN {X 0,Y 495.746,Z 386.73,A -85,B 0,C 180,E1 -6321.629,E2 -6321.629} C_VEL
LIN {X 0,Y 495.773,Z 386.733,A -85,B 0,C 180,E1 -6324.871,E2 -6324.871} C_VEL
LIN {X 0,Y 495.744,Z 386.725,A -85,B 0,C 180,E1 -6327.894,E2 -6327.894} C_VEL
LIN {X 0,Y 495.755,Z 386.733,A -85,B 0,C 180,E1 -6330.687,E2 -6330.687} C_VEL
LIN {X 0,Y 495.754,Z 386.722,A -85,B 0,C 180,E1 -6333.565,E2 -6333.565} C_VEL
LIN {X 0,Y 495.729,Z 386.737,A -85,B 0,C 180,E1 -6336.544,E2 -6336.544} C_VEL
LIN {X 0,Y 495.759,Z 386.727,A -85,B 0,C 180,E1 -6339.638,E2 -6339.638} C_VEL
LIN {X 0,Y 495.736,Z 386.733,A -85,B 0,C 180,E1 -6342.506,E2 -6342.506} C_VEL
LIN {X 0,Y 495.739,Z 386.73,A -85,B 0,C 180,E1 -6345.141,E2 -6345.141} C_VEL
LIN {X 0,Y 495.753,Z 386.73,A -85,B 0,C 180,E1 -6348.218,E2 -6348.218} C_VEL
LIN {X 0,Y 495.755,Z 386.729,A -85,B 0,C 180,E1 -6349.878,E2 -6349.878} C_VEL
LIN {X 0,Y 495.104,Z 386.813,A -85,B 0,C 180,E1 -6350.556,E2 -6350.556} C_VEL
LIN {X 0,Y 492.219,Z 387.174,A -85,B 0,C 180,E1 -6351.657,E2 -6351.657} C_VEL
LIN {X 0,Y 489.776,Z 387.477,A -85,B 0,C 180,E1 -6352.544,E2 -6352.544} C_VEL
LIN {X 0,Y 488.741,Z 387.605,A -85,B 0,C 180,E1 -6353.23,E2 -6353.23} C_VEL
LIN {X 0,Y 488.666,Z 387.613,A -85,B 0,C 180,E1 -6353.462,E2 -6353.462} C_VEL
LIN {X 0,Y 488.737,Z 387.61,A -85,B 0,C 180,E1 -6356.516,E2 -6356.516} C_VEL
LIN {X 0,Y 488.725,Z 387.604,A -85,B 0,C 180,E1 -6359.781,E2 -6359.781} C_VEL
LIN {X 0,Y 488.783,Z 387.834,A -85,B 0,C 180,E1 -6360.843,E2 -6360.843} C_VEL
LIN {X 0,Y 492.278,Z 403.454,A -85,B 0,C 180,E1 -6363.046,E2 -6363.046} C_VEL
LIN {X 0,Y 491.693,Z 425.638,A -85,B 0,C 180,E1 -6365.926,E2 -6365.926} C_VEL
LIN {X 0,Y 490.925,Z 448.11,A -85,B 0,C 180,E1 -6368.828,E2 -6368.828} C_VEL
LIN {X 0,Y 490.267,Z 470.22,A -85,B 0,C 180,E1 -6371.617,E2 -6371.617} C_VEL
LIN {X 0,Y 489.928,Z 488.136,A -85,B 0,C 180,E1 -6373.771,E2 -6373.771} C_VEL
LIN {X 0,Y 491.732,Z 501.284,A -85,B 0,C 180,E1 -6374.037,E2 -6374.037} C_VEL
LIN {X 0,Y 491.109,Z 599.002,A -85,B 0,C 180,E1 -6375.497,E2 -6375.497} C_VEL
LIN {X 0,Y 490.853,Z 612.193,A -85,B 0,C 180,E1 -6375.86,E2 -6375.86} C_VEL
LIN {X 0,Y 490.488,Z 624.654,A -85,B 0,C 180,E1 -6376.377,E2 -6376.377} C_VEL
LIN {X 0,Y 490.142,Z 636.444,A -85,B 0,C 180,E1 -6377.036,E2 -6377.036} C_VEL
LIN {X 0,Y 489.82,Z 646.901,A -85,B 0,C 180,E1 -6377.782,E2 -6377.782} C_VEL
LIN {X 0,Y 489.356,Z 657.385,A -85,B 0,C 180,E1 -6378.716,E2 -6378.716} C_VEL
LIN {X 0,Y 488.991,Z 665.981,A -85,B 0,C 180,E1 -6379.65,E2 -6379.65} C_VEL
LIN {X 0,Y 488.64,Z 675.345,A -85,B 0,C 180,E1 -6380.897,E2 -6380.897} C_VEL
LIN {X 0,Y 488.359,Z 682.792,A -85,B 0,C 180,E1 -6382.142,E2 -6382.142} C_VEL
LIN {X 0,Y 488.183,Z 688.771,A -85,B 0,C 180,E1 -6383.387,E2 -6383.387} C_VEL
LIN {X 0,Y 488.068,Z 693.504,A -85,B 0,C 180,E1 -6384.629,E2 -6384.629} C_VEL
LIN {X 0,Y 487.981,Z 697.129,A -85,B 0,C 180,E1 -6385.871,E2 -6385.871} C_VEL
LIN {X 0,Y 487.972,Z 698.995,A -85,B 0,C 180,E1 -6386.697,E2 -6386.697} C_VEL
LIN {X 0,Y 487.909,Z 700.425,A -85,B 0,C 180,E1 -6387.523,E2 -6387.523} C_VEL
LIN {X 0,Y 487.891,Z 701.426,A -85,B 0,C 180,E1 -6388.349,E2 -6388.349} C_VEL
LIN {X 0,Y 487.819,Z 702.283,A -85,B 0,C 180,E1 -6390,E2 -6390} C_VEL
LIN {X 0,Y 487.834,Z 702.096,A -85,B 0,C 180,E1 -6390.826,E2 -6390.826} C_VEL
LIN {X 0,Y 487.891,Z 701.511,A -85,B 0,C 180,E1 -6391.651,E2 -6391.651} C_VEL
LIN {X 0,Y 487.973,Z 699.179,A -85,B 0,C 180,E1 -6393.303,E2 -6393.303} C_VEL
LIN {X 0,Y 487.956,Z 696.308,A -85,B 0,C 180,E1 -6394.544,E2 -6394.544} C_VEL
LIN {X 0,Y 488.107,Z 692.406,A -85,B 0,C 180,E1 -6395.785,E2 -6395.785} C_VEL
LIN {X 0,Y 488.179,Z 687.355,A -85,B 0,C 180,E1 -6397.029,E2 -6397.029} C_VEL
